				IF CountAO = 0 THEN 
				// code for invalid object address	IOA : return command with invalid data . 
					stTxAsdu := stRxAsdu;
					IF stRxAsdu.info.objAddr = AODB[KK].aObj.obj.info.objAddr THEN
						stTxAsdu.ident.eCOT := eIEC870_COT_UNKNOWN_TYPE; // cause of transfer -> Wrong TYPE for this IoA .  
					ELSE
						stTxAsdu.ident.eCOT := eIEC870_COT_UNKNOWN_OBJECT_ADDRESS; // cause of transfer -> unknown IOA 
					END_IF
					stTxAsdu.ident.bPN :=  TRUE;					
					fbBuffer.TxAddObj(	putObj := stTxAsdu,
										buffer := stBuffer);
					IF NOT fbBuffer.bOk THEN
						// code for buffer overflow
						EXIT; 
					END_IF		 
					EXIT;
				END_IF
				
				
			C_SE_TC_1: // Télévaleurs	
				CountAO := 0 ; 
				FOR KK:=1 TO akuoPara.iAOnb DO 
					IF stRxAsdu.info.objAddr = AODB[KK].aObj.obj.info.objAddr THEN 
						CountAO := CountAO +1 ; ;
						F_iecCopyStreamToBuffer(ADR(nSCO_Val),SIZEOF(nSCO_Val),stRxAsdu.info.stream);
						// Get value of corresponding byte .
						TempData_bis := MesDword_Old[KK] XOR SHL(MesCmd_old[KK] ,AODB[KK].aObj.cfg.bitOffs )  ; 	// We set to zero here the bits that will be replaced
						TempData_bis := SHL(nSCO_Val AND Mask[KK] , AODB[KK].aObj.cfg.bitOffs) OR TempData_bis ;	// We insert the new bits 
			
						IF NOT IN_Local	THEN				// Permet de mettre à jour la commande que si pas en local
							MEMCPY( destAddr := memory+ULINT_TO_DWORD(AODB[KK].aObj.cfg.byteOffs) , srcAddr := ADR(TempData_bis) , n := nBytesRead[KK]);
							MesCmd := nSCO_Val AND Mask[KK] ;
					
						ELSE
							nSCO_Val := MesCmd_old[KK] ;
						END_IF	
					
						// create activation confirmation asdu
						stTxAsdu := stRxAsdu;
						F_iecCopyStreamToBufferByOffset(ADR(nSCO_Val),SIZEOF(nSCO_Val),0,stTxAsdu.info.stream);// Permet de mettre à jour que si pas en local	
						stTxAsdu.ident.eCOT := eIEC870_COT_ACT_CON; 				//cause of transfer -> activation confirmation
						
						IF IN_Local THEN
							stTxAsdu.ident.bPN :=  TRUE;
						ELSE 
							stTxAsdu.ident.bPN := FALSE;
						END_IF						
						
						fbBuffer.TxAddObj(	putObj := stTxAsdu,	buffer := stBuffer);
						IF NOT fbBuffer.bOk THEN
							// code for buffer overflow
							EXIT; 
						END_IF
						
						IF NOT IN_Local THEN
							stTxAsdu := stRxAsdu;
							stTxAsdu.ident.eCOT := eIEC870_COT_ACT_TERM; // cause of transfer -> activation termination
							stTxAsdu.ident.bPN := FALSE;
							fbBuffer.TxAddObj(	putObj := stTxAsdu,	buffer := stBuffer);
							IF NOT fbBuffer.bOk THEN
								// code for buffer overflow
								EXIT; 
							END_IF				
						END_IF
						
					END_IF
				END_FOR
				
				IF CountAO = 0 THEN 
				// code for invalid object address	IOA : return command with invalid data . 
					stTxAsdu := stRxAsdu;
					IF stRxAsdu.info.objAddr = AODB[KK].aObj.obj.info.objAddr THEN
						stTxAsdu.ident.eCOT := eIEC870_COT_UNKNOWN_TYPE; // cause of transfer -> Wrong TYPE for this IoA .  
					ELSE
						stTxAsdu.ident.eCOT := eIEC870_COT_UNKNOWN_OBJECT_ADDRESS; // cause of transfer -> unknown IOA 
					END_IF
					stTxAsdu.ident.bPN :=  TRUE;					
					fbBuffer.TxAddObj(	putObj := stTxAsdu,
										buffer := stBuffer);
					IF NOT fbBuffer.bOk THEN
						// code for buffer overflow
						EXIT; 
					END_IF		 
					EXIT;
				END_IF
			
			C_CS_NA_1: 
				// clock synchronisation
				F_iecCopyStreamToBuffer(ADR(tActTime),SIZEOF(tActTime),stRxAsdu.info.stream);	
	
				// create clock sync confirmation asdu
				stTxAsdu := stRXAsdu;
				stTxAsdu.ident.eCOT := eIEC870_COT_ACT_CON; // cause of transfer -> activation confirmation
				fbBuffer.TxAddObj(	putObj := stTxAsdu,
									buffer := stBuffer);
				IF NOT fbBuffer.bOk THEN
					// code for buffer overflow
					EXIT; 
				END_IF
				// set local computer time
				fbsetLocalTime( START	:= TRUE,
								NETID	:= '', 
								TIMESTR	:= CP56Time2a_TO_SYSTEMTIME(tActTime,20) );
				fbsetLocalTime( START	:= FALSE);
		ELSE
				// code for invalid asdu types 
				stTxAsdu := stRxAsdu;
				stTxAsdu.ident.eCOT := eIEC870_COT_UNKNOWN_TYPE; // cause of transfer -> unknown Type ASDU 
				stTxAsdu.ident.bPN :=  TRUE;					
				fbBuffer.TxAddObj(	putObj := stTxAsdu,
									buffer := stBuffer);
				IF NOT fbBuffer.bOk THEN
					// code for buffer overflow
					EXIT; 
				END_IF		
			
			EXIT;
		END_CASE
	END_IF

UNTIL NOT fbBuffer.bOk // RX fifo is empty
END_REPEAT
END_METHOD

END_FUNCTION_BLOCK

// ---- 00_FunctionsBlocks/Common/AlarmManagement/FB_DetectFlicker.TcPOU
FUNCTION_BLOCK FB_DetectFlicker
// Detect if a booleean variable is flickering 

VAR_INPUT
	IN_VAR			: BOOL;						// Boolean input to analyze
	IN_Window		: TIME := T#5S;				// Time Window during which I check the number of value change
	IN_Count		: UINT;						// Maximum number of change for the tiume duration 

END_VAR
VAR_OUTPUT
	OUT_bFlicker		: BOOL;					// Value is considered as flickering
END_VAR
VAR
	COUNT 			: CTU ; 
	TON				: TON ; 
END_VAR

TON(IN:= TRUE , PT:= IN_Window ) ; 

IF COUNT.CV > IN_Count THEN 
	OUT_bFlicker := TRUE ; 
ELSIF COUNT.CV < IN_Count AND TON.Q THEN  
	OUT_bFlicker := FALSE ; 
END_IF	
	
COUNT(CU:= IN_VAR , PV:= 1000 , RESET:=TON.Q)  ; 

IF TON.Q THEN 
	TON(IN:= FALSE ) ; 
END_IF

END_FUNCTION_BLOCK

// ---- 00_FunctionsBlocks/Beckhoff/Communication/ModbusRTU/Sample_ModbusRTU.TcPOU
PROGRAM Sample_ModbusRTU
VAR
	ModbusRTU				: FB_ModbusRTU;
	MesBlock				: ARRAY[1..8] OF ARRAY[1..120] OF WORD;	
	AX_Addr					: ARRAY[1..8] OF UINT 	:= [1,		1,		1,		1,		1, 		1, 		1, 		1];
	AX_Qty					: ARRAY[1..8] OF UINT	:= [1,		1,		1,		1,		1, 		1, 		1, 		1];
	AX_UnitId				: ARRAY[1..8] OF BYTE	:= [1,		1,		1,		1,		1, 		1, 		1, 		1];
	AX_Function				: ARRAY[1..8] OF UINT	:= [1,		2,		3,		4,		5, 	 	6, 	 	15, 	16];	
	AX_Priority				: ARRAY[1..8] OF UINT	:= [1,		1,		1,		1,		1, 	 	1, 	 	1, 		1 ];
	AX_bStart				: ARRAY[1..8] OF BOOL;
	MbStruct				: ARRAY[1..8] OF Struct_InputRTU;	
	
	KK: INT;
END_VAR

ModbusRTU();

FOR KK := 1 TO 8 DO 
	MbStruct[KK].InBuffer := ADR(MesBlock[KK]);
	MbStruct[KK].InFunction := AX_Function[KK];
	MbStruct[KK].InQuantity := AX_Qty[KK];
	MbStruct[KK].InStartAddr := AX_Addr[KK];
	MbStruct[KK].InUnitID := AX_UnitId[KK];
END_FOR


IF CalLocalTimeStruct.wSecond MOD 5 = 0 THEN
	FOR KK := 1 TO 8 DO
		IF AX_bStart[KK] THEN
			ModbusRTU.M_AddAction_FIFO(InStruct := MbStruct[KK], InPriority := AX_Priority[KK]);
		END_IF
	END_FOR
	
END_IF

END_PROGRAM

// ---- 00_FunctionsBlocks/Beckhoff/Communication/ModbusTCP/FB_ModbusReadCoils.TcPOU
FUNCTION_BLOCK FB_ModbusReadCoils
////////////////// 
// Read Modbus TCP/IP on Rising Edge of Trigger ClockRead. Returns alarm and stop modbus Read after three consecutive Modbus attempts that failed. 
//////////////////

VAR_INPUT
	
	// Modbus ReadRegs FB inputs
	pDestAddr 	: POINTER TO BYTE ; // Pointer to variable in which the read data have to be stored
	sIPAddr 	: STRING(15);		// Modbus server device IP adress
	tTimeout 	: TIME;				// Timeout
	nTcpPort 	: UINT;
	nQuantity 	: WORD;				// Quantity of words to be read
	nMBAddr 	: WORD ;			// Starting Register adress
	
	cbLength 	: UDINT;			// Length of variable to host the read data
	nUnitID 	: BYTE;				// Unit ID in case of serial connexion after modbus server. Usually equals to 1
	
	ClockRead	: BOOL; 			// Rising Edge Modbus Trigger
	Reset		: BOOL; 			// Reset Trigger to clean alarm and counter.
	
END_VAR

VAR_OUTPUT
	ErrorId			: UDINT;	// Error Id returned by FB ( see ADS error Code ) . 
	
	Busy			: BOOL ;	// FB busy to proceed command
	ModbusReadAlarm	: BOOL; 	// Alarm if three modbus attempt failed.
	OUT_NbRead		: UDINT;
END_VAR

VAR
	R_TRIG 				: R_TRIG; 			// Rising edge detection for the trigger.
	FB_MBReadCoils 		: FB_MBReadCoils; 	// Multiple registers reading
	
	Step				: INT; 				// Grafcet step
	AlarmCounter		: INT; 				// Alarm Counter. Incremennted if modbus errOR  Alarm if counter =3 , resetable.  

	
END_VAR

// ALARM MANAGEMENT //

	IF AlarmCounter=3 THEN 
		ModbusReadAlarm 	:=TRUE;
		
	ELSE
		ModbusReadAlarm := FALSE;
		ErrorId			:= 0;
		
	END_IF


// MODBUS SEQUENCE //
CASE Step OF 
	0:
		R_TRIG(CLK :=ClockRead);
		
		IF R_TRIG.Q THEN 
			Step :=1;
			Busy := TRUE;
			OUT_NbRead := 0;
		END_IF
	1:
	   FB_MBReadCoils(
	  			sIPAddr:= sIPAddr , 
				nTCPPort:= nTcpPort ,
				nUnitID:= nUnitID,
				nQuantity:= nQuantity,
				nMBAddr:= nMBAddr, 
				cbLength:= cbLength, 
				pDestAddr:= pDestAddr, 
				bExecute:= TRUE,
				tTimeout:= tTimeout,
				cbRead => OUT_NbRead
				);
				
		IF NOT FB_MBReadCoils.bBusy AND NOT FB_MBReadCoils.bError THEN
			FB_MBReadCoils(bExecute:= FALSE);
			AlarmCounter	:=0; // Reset counter after successful modbus read. 
			Step 			:=0;
			Busy := FALSE;
		ELSIF NOT FB_MBReadCoils.bBusy AND FB_MBReadCoils.bError THEN
			FB_MBReadCoils(bExecute:= FALSE);
			AlarmCounter 	:= MIN(AlarmCounter+1,3) ; 
			ErrorId			 :=FB_MBReadCoils.nErrId;
			Step 			:=0;
			Busy := FALSE;
		END_IF
		
END_CASE

// RESET //
	IF Reset THEN 
			AlarmCounter 		:= 0 ; 
			ErrorId 			:= 0 ; 
			ModbusReadAlarm 	:=FALSE;
			Reset 				:= FALSE;
			FB_MBReadCoils		(bExecute := FALSE);
	END_IF

// BUSY //

END_FUNCTION_BLOCK

// ---- 00_FunctionsBlocks/Beckhoff/Communication/ModbusTCP/FB_ModbusReadInput.TcPOU
FUNCTION_BLOCK FB_ModbusReadInput
////////////////// 
// Read Modbus TCP/IP on Rising Edge of Trigger ClockRead. Returns alarm and stop modbus Read after three consecutive Modbus attempts that failed. 
//////////////////

VAR_INPUT
	
	// Modbus ReadRegs FB inputs
	pDestAddr 	: POINTER TO BYTE ; // Pointer to variable in which the read data have to be stored
	sIPAddr 	: STRING(15);		// Modbus server device IP adress
	tTimeout 	: TIME;				// Timeout
	nTcpPort 	: UINT;
	nQuantity 	: WORD;				// Quantity of words to be read
	nMBAddr 	: WORD ;			// Starting Register adress
	
	cbLength 	: UDINT;			// Length of variable to host the read data
	nUnitID 	: BYTE;				// Unit ID in case of serial connexion after modbus server. Usually equals to 1
	
	ClockRead	: BOOL; 			// Rising Edge Modbus Trigger
	Reset		: BOOL; 			// Reset Trigger to clean alarm and counter.
	
END_VAR

VAR_OUTPUT
	ErrorId			: UDINT;	// Error Id returned by FB ( see ADS error Code ) . 
	
	Busy			: BOOL ;	// FB busy to proceed command
	ModbusReadAlarm	: BOOL; 	// Alarm if three modbus attempt failed.
	OUT_NbRead		: UDINT;
END_VAR

VAR
	R_TRIG 				: R_TRIG; 			// Rising edge detection for the trigger.
	FB_MBReadInputs 		: FB_MBReadInputs; 	// Multiple registers reading
	
	Step				: INT; 				// Grafcet step
	AlarmCounter		: INT; 				// Alarm Counter. Incremennted if modbus errOR  Alarm if counter =3 , resetable.  

	
END_VAR

// ALARM MANAGEMENT //

	IF AlarmCounter=3 THEN 
		ModbusReadAlarm 	:=TRUE;
		
	ELSE
		ModbusReadAlarm := FALSE;
		ErrorId			:= 0;
		
	END_IF


// MODBUS SEQUENCE //
CASE Step OF 
	0:
		R_TRIG(CLK :=ClockRead);
		
		IF R_TRIG.Q THEN 
			Step :=1;
			Busy := TRUE;
			OUT_NbRead := 0;
		END_IF
	1:
	   FB_MBReadInputs(
	  			sIPAddr:= sIPAddr , 
				nTCPPort:= nTcpPort ,
				nUnitID:= nUnitID,
				nQuantity:= nQuantity,
				nMBAddr:= nMBAddr, 
				cbLength:= cbLength, 
				pDestAddr:= pDestAddr, 
				bExecute:= TRUE,
				tTimeout:= tTimeout,
				cbRead => OUT_NbRead
				);
				
		IF NOT FB_MBReadInputs.bBusy AND NOT FB_MBReadInputs.bError THEN
			FB_MBReadInputs(bExecute:= FALSE);
			AlarmCounter	:=0; // Reset counter after successful modbus read. 
			Step 			:=0;
			Busy := FALSE;
		ELSIF NOT FB_MBReadInputs.bBusy AND FB_MBReadInputs.bError THEN
			FB_MBReadInputs(bExecute:= FALSE);
			AlarmCounter 	:= MIN(AlarmCounter+1,3) ; 
			ErrorId			 :=FB_MBReadInputs.nErrId;
			Step 			:=0;
			Busy := FALSE;
		END_IF
		
END_CASE

// RESET //
	IF Reset THEN 
			AlarmCounter 		:= 0 ; 
			ErrorId 			:= 0 ; 
			ModbusReadAlarm 	:=FALSE;
			Reset 				:= FALSE;
			FB_MBReadInputs		(bExecute := FALSE);
	END_IF

// BUSY //

END_FUNCTION_BLOCK

// ---- 00_FunctionsBlocks/Beckhoff/Communication/ModbusTCP/FB_ModbusWriteMultipleCoils.TcPOU
FUNCTION_BLOCK FB_ModbusWriteMultipleCoils
////////////////// 
// Write Modbus TCP/IP on Rising Edge of Trigger WriteCommAND  Returns alarm and stop modbus Read after three consecutive Modbus attempts that failed.
// Write two registers 
//////////////////
VAR_INPUT
	// Modbus ReadRegs FB inputs

	pSrcAddr			: POINTER TO BYTE ;
	sIPAddr 			: STRING(15);
	tTimeout 			: TIME;
	nTCPport			: UINT:= 502;		// TCP Port
	nMBAddr 			: WORD ;
	cbLength 			: UDINT ;
	nQuantity			: BYTE ;
	nUnitID 			: BYTE;
	WriteCmd 			: BOOL; 					// Rising Edge Trigger for sending modbus request
	
	Reset				: BOOL; 					// Reset Trigger to clean alarm and counter	
	
END_VAR


VAR_OUTPUT
	ErrorId				: UDINT; 			// Erreur ID returned by FB modbus. Updated every time on error occurs. 
	
	Completed			: BOOL ;			// Modbus Writing is completed 
	Busy				: BOOL ; 			// FB busy to proceed command
	ModbusWriteAlarm	: BOOL; 			// Alarm if three modbus attempt failed.
	
END_VAR
VAR
	R_TRIG 				: R_TRIG; 				// Rising edge detection for the trigger.
	FB_MBWriteCoils		: FB_MBWriteCoils; 		// Multiple registers reading
	
	Step				: INT; 					// Grafcet step
	AlarmCounter		: INT; 					// Alarm Counter. Incremennted if modbus errOR  Alarm if counter =3 , resetable.  
END_VAR

Completed 				:= FALSE ;

// ALARM MANAGEMENT //
IF AlarmCounter=3 THEN
	ModbusWriteAlarm 	:=TRUE;
	
ELSE
	ModbusWriteAlarm 	:= FALSE;
	ErrorId				:= 0;
	
END_IF
	
// MODBUS SEQUENCE //
	CASE Step OF 
		0:
			R_TRIG(CLK :=WriteCmd);
			IF R_TRIG.Q THEN 
				Step :=1;
			END_IF
			
		1:
		   FB_MBWriteCoils(
					sIPAddr:= sIPAddr , 
					nTCPPort:= nTCPport ,
					nUnitID:= nUnitID,
					nQuantity:= nQuantity,
					nMBAddr:= nMBAddr, 
					cbLength:= cbLength, 
					pSrcAddr:= pSrcAddr, 
					bExecute:= TRUE,
					tTimeout:= tTimeout
					);
					
			IF NOT FB_MBWriteCoils.bBusy AND NOT FB_MBWriteCoils.bError THEN
				FB_MBWriteCoils(bExecute:= FALSE);
				AlarmCounter		:=0; // Reset counter after successful modbus read. 
				Step 				:=0;
				Completed 			:= TRUE ;
				
			ELSIF NOT FB_MBWriteCoils.bBusy AND FB_MBWriteCoils.bError THEN
				FB_MBWriteCoils(bExecute:= FALSE);
				AlarmCounter 		:=MIN(AlarmCounter+1,3) ; 
				ErrorId			 	:=FB_MBWriteCoils.nErrId;
				Step 				:=0;
				
			END_IF
			
	END_CASE

// RESET //	
	IF Reset THEN 
			AlarmCounter 	:= 0 ; 
			ErrorId 		:= 0 ; 
	END_IF	
	
// BUSY //
	Busy 					:= FB_MBWriteCoils.bBusy ;

END_FUNCTION_BLOCK

// ---- 00_FunctionsBlocks/Beckhoff/Communication/ModbusTCP/FB_ModbusWriteSingleCoil.TcPOU
FUNCTION_BLOCK FB_ModbusWriteSingleCoil
////////////////// 
// Write Modbus TCP/IP on Rising Edge of Trigger WriteCommAND  Returns alarm and stop modbus Read after three consecutive Modbus attempts that failed.
// Write two registers 
//////////////////
VAR_INPUT
	// Modbus ReadRegs FB inputs
	bValue 				: BOOL;
	sIPAddr 			: STRING(15);
	tTimeout 			: TIME;
	nTCPport			: UINT:= 502;		// TCP Port
	nMBAddr 			: WORD ;
	nUnitID 			: BYTE;
	WriteCmd 			: BOOL; 					// Rising Edge Trigger for sending modbus request
	
	Reset				: BOOL; 					// Reset Trigger to clean alarm and counter	
	
END_VAR


VAR_OUTPUT
	ErrorId				: UDINT; 			// Erreur ID returned by FB modbus. Updated every time on error occurs. 
	
	Completed			: BOOL ;			// Modbus Writing is completed 
	Busy				: BOOL ; 			// FB busy to proceed command
	ModbusWriteAlarm	: BOOL; 			// Alarm if three modbus attempt failed.
	
END_VAR
VAR
	R_TRIG 				: R_TRIG; 				// Rising edge detection for the trigger.
	FB_MBWriteSingleCoil: FB_MBWriteSingleCoil; 		// Multiple registers reading
	
	Step				: INT; 					// Grafcet step
	AlarmCounter		: INT; 					// Alarm Counter. Incremennted if modbus errOR  Alarm if counter =3 , resetable.  
	wValue				: WORD;
END_VAR

Completed 				:= FALSE ;

// ALARM MANAGEMENT //
IF AlarmCounter=3 THEN
	ModbusWriteAlarm 	:=TRUE;
	
ELSE
	ModbusWriteAlarm 	:= FALSE;
	ErrorId				:= 0;
	
END_IF

IF bValue THEN
	wValue := 16#FF00;
ELSE
	wValue := 16#0000;
END_IF
	
// MODBUS SEQUENCE //
	CASE Step OF 
		0:
			R_TRIG(CLK :=WriteCmd);
			IF R_TRIG.Q THEN 
				Step :=1;
			END_IF
			
		1:
		   FB_MBWriteSingleCoil
			(
				sIPAddr:= sIPAddr ,
				nValue := wValue,
				nTCPPort:= nTCPport ,
				nUnitID:= nUnitID,
				nMBAddr:= nMBAddr, 
				bExecute:= TRUE,
				tTimeout:= tTimeout
			);
					
			IF NOT FB_MBWriteSingleCoil.bBusy AND NOT FB_MBWriteSingleCoil.bError THEN
				FB_MBWriteSingleCoil(bExecute:= FALSE);
				AlarmCounter		:=0; // Reset counter after successful modbus read. 
				Step 				:=0;
				Completed 			:= TRUE ;
				
			ELSIF NOT FB_MBWriteSingleCoil.bBusy AND FB_MBWriteSingleCoil.bError THEN
				FB_MBWriteSingleCoil(bExecute:= FALSE);
				AlarmCounter 		:=MIN(AlarmCounter+1,3) ; 
				ErrorId			 	:=FB_MBWriteSingleCoil.nErrId;
				Step 				:=0;
				
			END_IF
			
	END_CASE

// RESET //	
	IF Reset THEN 
			AlarmCounter 	:= 0 ; 
			ErrorId 		:= 0 ; 
	END_IF	
	
// BUSY //
	Busy 					:= FB_MBWriteSingleCoil.bBusy ;

END_FUNCTION_BLOCK

// ---- 00_FunctionsBlocks/Beckhoff/Communication/ModbusTCP/FB_ModbusWriteSingleRegister.TcPOU
FUNCTION_BLOCK FB_ModbusWriteSingleRegister
////////////////// 
// Write Modbus TCP/IP on Rising Edge of Trigger WriteCommAND  Returns alarm and stop modbus Read after three consecutive Modbus attempts that failed.
// Write two registers 
//////////////////
VAR_INPUT
	// Modbus ReadRegs FB inputs

	InputWord			: WORD ;
	sIPAddr 			: STRING(15);
	tTimeout 			: TIME;
	nTCPport			: UINT:= 502;		// TCP Port
	nMBAddr 			: WORD ;
	cbLength 			: UDINT ;
	nQuantity			: BYTE ;
	nUnitID 			: BYTE;
	WriteCmd 			: BOOL; 					// Rising Edge Trigger for sending modbus request
	
	Reset				: BOOL; 					// Reset Trigger to clean alarm and counter	
	
END_VAR


VAR_OUTPUT
	ErrorId						: UDINT; 			// Erreur ID returned by FB modbus. Updated every time on error occurs. 
	                    		
	Completed					: BOOL ;			// Modbus Writing is completed 
	Busy						: BOOL ; 			// FB busy to proceed command
	ModbusWriteAlarm			: BOOL; 			// Alarm if three modbus attempt failed.
	
END_VAR
VAR
	R_TRIG 						: R_TRIG; 				// Rising edge detection for the trigger.
	MBWriteSingleReg 		: FB_MBWriteSingleReg; 		// Multiple registers reading
	
	Step						: INT; 					// Grafcet step
	AlarmCounter				: INT; 					// Alarm Counter. Incremennted if modbus errOR  Alarm if counter =3 , resetable.  
END_VAR

Completed 				:= FALSE ;

// ALARM MANAGEMENT //
IF AlarmCounter=3 THEN
	ModbusWriteAlarm 	:=TRUE;
	
ELSE
	ModbusWriteAlarm 	:= FALSE;
	ErrorId				:= 0;
	
END_IF
	
// MODBUS SEQUENCE //
	CASE Step OF 
		0:
			R_TRIG(CLK :=WriteCmd);
			IF R_TRIG.Q THEN 
				Step :=1;
			END_IF
			
		1:
		   MBWriteSingleReg(
			   		nValue := InputWord,
					sIPAddr:= sIPAddr , 
					nTCPPort:= nTCPport ,
					nUnitID:= nUnitID,
					nMBAddr:= nMBAddr, 
					bExecute:= TRUE,
					tTimeout:= tTimeout
					);
					
			IF NOT MBWriteSingleReg.bBusy AND NOT MBWriteSingleReg.bError THEN
				MBWriteSingleReg(bExecute:= FALSE);
				AlarmCounter		:=0; // Reset counter after successful modbus read. 
				Step 				:=0;
				Completed 			:= TRUE ;
				
			ELSIF NOT MBWriteSingleReg.bBusy AND MBWriteSingleReg.bError THEN
				MBWriteSingleReg(bExecute:= FALSE);
				AlarmCounter 		:=MIN(AlarmCounter+1,3) ; 
				ErrorId			 	:=MBWriteSingleReg.nErrId;
				Step 				:=0;
				
			END_IF
			
	END_CASE

// RESET //	
	IF Reset THEN 
			AlarmCounter 	:= 0 ; 
			ErrorId 		:= 0 ; 
			Reset			:= FALSE;
			MBWriteSingleReg(bExecute := FALSE);
	END_IF	
	
// BUSY //
	Busy 					:= MBWriteSingleReg.bBusy ;

END_FUNCTION_BLOCK

// ---- 00_FunctionsBlocks/Beckhoff/Database/CheckConfig.TcPOU
PROGRAM CheckConfig
VAR_INPUT
		IN_Start				: BOOL := TRUE;
		ParamInitWait			: TIME := T#5S;
END_VAR
VAR_OUTPUT
		OUT_aDBConfig         		: ARRAY[0..MAX_CONFIGURATIONS] OF ST_ConfigDB;
		OUT_Busy					: BOOL;
		OUT_Error					: BOOL;
		OUT_Result					: INT;
END_VAR
VAR
	// CheckConfig    
		TON_CheckConfig				: TON;      		
		TrigCheckConfig				: R_TRIG;
		TrigInit					: F_TRIG;
		RS_CheckConfig				: RS;
		                    		
		ConfigTcDBSrvEvt  			: FB_ConfigTcDBSrvEvt(sNetId := '', tTimeout:=T#5S);
		                    		
		aAutoGrpConfig    			: ARRAY[0..MAX_CONFIGURATIONS] OF ST_ConfigAutoLogGrp;
		AX_NameBase					: ARRAY[0..MAX_CONFIGURATIONS] OF T_MaxString;
		AX_hDBID					: ARRAY[0..MAX_CONFIGURATIONS] OF BOOL;
		AX_hDBIDNull				: ARRAY[0..MAX_CONFIGURATIONS] OF BOOL;
		                    		
		nDbCount          			: UDINT;
		nAutoGrpCount     			: UDINT;

		KK : UDINT;
END_VAR

TON_CheckConfig(IN := IN_Start, PT := ParamInitWait);

TrigCheckConfig(CLK := TON_CheckConfig.Q);
RS_CheckConfig(SET := TrigCheckConfig.Q);
IF TrigCheckConfig.Q THEN
	IN_Start := FALSE;
	OUT_Result := 0;
END_IF
IF RS_CheckConfig.Q1 THEN
	
	OUT_Busy := TRUE;
	IF ConfigTcDBSrvEvt.Read(pDBConfig := ADR(OUT_aDBConfig), cbDBConfig := SIZEOF(OUT_aDBConfig), pAutologGrpConfig := ADR(aAutoGrpConfig),
			cbAutoLogGrpConfig := SIZEOF(aAutoGrpConfig),pDBCount := ADR(nDbCount),pAutoLogGrpCount := ADR(nAutoGrpCount)) THEN
		
		IF ConfigTcDBSrvEvt.bError THEN
			OUT_Result := -1;
		ELSE
			FOR KK := 0 TO MAX_CONFIGURATIONS DO
				AX_hDBID[OUT_aDBConfig[KK].hDBID] := OUT_aDBConfig[KK].hDBID <> 0;
				AX_NameBase[KK] :=  OUT_aDBConfig[KK].sName;
			END_FOR
			OUT_Result := 1;
		END_IF  
		RS_CheckConfig(RESET1 := TRUE);
		RS_CheckConfig(RESET1 := FALSE);
		OUT_Busy := FALSE;
		
	END_IF
END_IF

END_PROGRAM

// ---- 00_FunctionsBlocks/Beckhoff/Database/Firebird/Firebird_CreateTables.TcPOU
PROGRAM Firebird_CreateTables
VAR_INPUT
	IN_Start				: BOOL;
	IN_TableNames			: ARRAY[1.. CstNbTables] OF STRING;
	IN_hDBID         		: UDINT;	
END_VAR
VAR_OUTPUT
	OUT_Error				: BOOL;
	OUT_Busy				: BOOL;
	OUT_Result				: INT;
END_VAR
VAR
	Etape					: UINT;
	
	TrigStart				: R_TRIG;
	RsStart					: RS;
	bCreateTable			: BOOL;
	TrigCreateTable			: R_TRIG;
	RsCreateTable			: RS;
	PLCDBCreateEvt 			: FB_PLCDBCreateEvt(sNetID := '', tTimeout := T#5S);
	FirebirdConf			: T_DBConfig_Odbc;
	sExtension				: STRING:= '.db';
	tcMessage    	 		: I_TcMessage;
	
	AX_ColArray				: ARRAY[0..3] OF ST_ColumnInfo;
	
	NumTable				: UINT := 1;
	KK						: UDINT;
END_VAR


AX_ColArray[0].sName := 'TimeStamp';     	AX_ColArray[0].eType := E_ColumnType.DateTime;   	AX_ColArray[0].nLength := 4;    
AX_ColArray[1].sName := 'TimeStamp_Ms';    	AX_ColArray[1].eType := E_ColumnType.Integer;    	AX_ColArray[1].nLength := 4;
AX_ColArray[2].sName := 'ParentId';   		AX_ColArray[2].eType := E_ColumnType.Integer;   	AX_ColArray[2].nLength := 4;
AX_ColArray[3].sName := 'Value';   			AX_ColArray[3].eType := E_ColumnType.Float;   		AX_ColArray[3].nLength := 8;


TrigCreateTable(CLK := IN_Start);
RsCreateTable(SET:= TrigCreateTable.Q);

IF RsCreateTable.Q1 THEN
	OUT_Busy := TRUE;
	IF NumTable <= CstNbTables THEN
		IF PLCDBCreateEvt.Table(hDBID := IN_hDBID, sTableName := IN_TableNames[NumTable],  pTableCfg := ADR(AX_ColArray), cbTableCfg := SIZEOF(AX_ColArray)  ) THEN
			IF PLCDBCreateEvt.bError THEN
				Etape := 255;
				OUT_Error := TRUE;
				OUT_Result := -2;
			ELSE
				IF Numtable = CstNbTables THEN
					IN_Start := FALSE;
					Etape := 0;
					RsCreateTable(RESET1 := TRUE);
					RsCreateTable(RESET1 := FALSE);	
					bCreateTable := FALSE;
					OUT_Result := 1;	
					TrigStart(CLK := FALSE);
					OUT_Busy := FALSE;	
					OUT_Error := FALSE;
					OUT_Result := 1;
				ELSE
					NumTable := NumTable + 1;		
				END_IF
			END_IF
		END_IF
	END_IF
END_IF

IF Etape = 255 THEN
	Etape := 0;
	bCreateTable := FALSE;
	IN_Start := FALSE;
	OUT_Busy := FALSE;	
	RsCreateTable(RESET1 := TRUE);
	RsCreateTable(RESET1 := FALSE);
END_IF

END_PROGRAM

// ---- 00_FunctionsBlocks/Beckhoff/Database/Firebird/Firebird_InsertBuffer.TcPOU
FUNCTION_BLOCK Firebird_InsertBuffer
// Fonctionnement : Tableau de 2000 structures en input. Dès qu'on atteint 1000 structures remplies, décalage de l'espace mémoire
// pour en 1 temps de cycle pour ne pas perdre de données sur le transfert.
VAR CONSTANT
	//CstNbLigneBuffer					: UINT:= 500;
	CstNbLigneBufferMax	 				: DINT:= 1000;
                            			
END_VAR                     			
                            			
VAR_INPUT                   			
	NomTable							: STRING(255) := 'Table100ms';
	IN_Reset							: BOOL;
	IN_Hdbid							: DINT;
	ParamTimeOut						: TIME := T#10s;
END_VAR                     			
                            			
VAR_OUTPUT                  			
	OUT_Error							: BOOL;
	OUT_Busy							: BOOL;
	OUT_Result							: INT;
	Out_Connected						: BOOL;
END_VAR                     			
                            			
VAR                         		
	Etape_main							: UINT:=2;	
	ETAPE								: UINT;
		CstNbLigneBuffer					: UINT:= 500;
	FTrig_TP_Retry						: F_TRIG;                        			
	TrigReset							: R_TRIG;
	TON_Watchdog						: TON ;
	TP_Retry							: TP;
	Tmp_Nb_Buffer						: DINT;
    //myStruct      						: ARRAY[1..CstNbLigneBuffer] OF St_DataHisto;
	//myStructMax    						: ARRAY[1..CstNbLigneBufferMax] OF St_DataHisto;
	StructNull							: St_DataHisto;
                            			
    SQLDatabase1						: FB_SQLDatabaseEvt('',T#10S);
    SQLDatabase2						: FB_SQLDatabaseEvt('',T#10S);
	SQLCommand1							: FB_SQLCommandEvt('',T#10S);
	SQLCommand2							: FB_SQLCommandEvt('',T#10S);
	
	bConnected							: BOOL;              	        	
                            			
	TrameValues							: T_MaxString := ' ([Timestamp],[ParentId],[Value])';
	pPosRequete							: DINT;                		
	RequeteFinale						: ARRAY[1..10000] OF STRING(1000);	
	RequeteFinaleNull					: ARRAY [1..10000] OF STRING(1000);
	
	sTimeStamp							: STRING(255);  
	RequeteEntete						: STRING(1000);
	sInsertValue						: STRING(1000);
	Format								: FB_FormatString;
	                			
	NbElemBuffer						: DINT;
	KK									: DINT;
	                    				
	CmdStart							: BOOL;
	TrigRestartMaxReached				: R_TRIG;
	TrigCmdExec							: R_TRIG;
	TrigStart							: R_TRIG;
	RsStart								: RS;
	                        			
	// AlarmManagement      			
		bBufferMaxFull 					: BOOL;        		
		bInStructNull					: BOOL;
		
	// CONNECT	
		TrigStartConnect				: R_TRIG;	
		RsStartConnect					: RS;
	// DISCONNECT
		TrigStartDisconnect				: R_TRIG;
		RsStartDisconnect				: RS;

		bReconnect						: BOOL;
		FTrig_bReconnect				: F_TRIG;
			
	MesAlarm: BOOL;
	TrigWatchdog : R_TRIG;
	bTest: BOOL;
	FIFO						: FB_DBDatasetFifo_1min;
END_VAR    

VAR_IN_OUT
	
END_VAR


//CmdStart := FIFO.nCount>= CstNbLigneBuffer AND NOT FTrig_TP_Retry.Q;
CmdStart := FIFO.nCount >= 0 AND NOT FTrig_TP_Retry.Q;


TP_Retry(IN := FIFO.nCount >= CstNbLigneBufferMax AND NOT TP_Retry.Q, PT := T#3S);
FTrig_TP_Retry(CLK := TP_Retry.Q);

TrigReset(CLK := IN_Reset OR TON_Watchdog.Q);
IF TrigReset.Q THEN
	FIFO.A_Reset();
END_IF

TrigStart(CLK := CmdStart);
IF TrigStart.Q THEN
	ETAPE := 1;
END_IF


RsStart(SET := TrigStart.Q);
IF RsStart.Q1 THEN
	RequeteEntete :=  concat(concat(' INSERT INTO "',NomTable),'" ');
END_IF
		
CASE ETAPE OF
		
	1: // CONNECTED
		IF SQLDatabase1.CreateCmd(pSQLCommand := ADR(SQLCommand1)) THEN 
			IF NOT SQLDatabase1.bError THEN
				MEMCPY(srcAddr:= ADR(RequeteEntete), destAddr := ADR(requeteFinale), n:= SIZEOF(RequeteEntete));
				pPosRequete := LEN(STR := RequeteEntete);
				Tmp_Nb_Buffer :=UDINT_TO_DINT(FIFO.nCount -1);
				FOR KK:= 1 TO MIN(Tmp_Nb_Buffer,CstNbLigneBuffer-1) DO
					fifo.A_Get();
					sTimeStamp	:=  SYSTEMTIME_TO_STRING(fifo.Out.Timestamp);
					Format(sFormat := 'select $'%s$',%.4d,%5.2f FROM RDB$$DATABASE UNION ALL ', arg1 := F_STRING(sTimeStamp),arg2:= F_DINT(fifo.out.ParentId), arg3:= F_LREAL(fifo.out.Value), arg5:= F_STRING(NomTable), sOut=>sInsertValue);
					MEMCPY(srcAddr:= ADR(sInsertValue), destAddr := ADR(requeteFinale)+DINT_TO_DWORD(pPosRequete), n:= SIZEOF(sInsertValue));
					pPosRequete:= pPosRequete + LEN(STR := sInsertValue);
					fifo.A_Remove();
				END_FOR
				fifo.A_Get();
				sTimeStamp	:= SYSTEMTIME_TO_STRING(fifo.Out.Timestamp);
				Format(sFormat := 'select $'%s$',%.4d,%5.2f FROM RDB$$DATABASE;', arg1 := F_STRING(sTimeStamp),arg2:= F_DINT(fifo.out.ParentId), arg3:= F_LREAL(fifo.out.Value), sOut=>sInsertValue);
				MEMCPY(srcAddr:= ADR(sInsertValue), destAddr := ADR(requeteFinale)+DINT_TO_DWORD(pPosRequete), n:= SIZEOF(sInsertValue));
				fifo.A_Remove();
				IF Tmp_Nb_Buffer > 0 THEN
					ETAPE := Etape_main;
				END_IF
			ELSIF SQLDatabase1.bError THEN
				ETAPE := 255;
			END_IF
		END_IF
	2:

		IF SQLCommand1.Execute(pSQLCmd := ADR(RequeteFinale), cbSQLCmd := SIZEOF(Requetefinale))THEN
			
			IF  NOT SQLCommand1.bError THEN
				ETAPE := 4;
			ELSIF SQLCommand1.bError THEN
				ETAPE := 255;
			END_IF
		END_IF

	4:
		IF NOT SQLDatabase1.bError THEN
			
			RequeteFinale := RequeteFinaleNull;
			
			//RequeteFinale := '';
			Tmp_Nb_Buffer := MIN(UDINT_TO_DINT(FIFO.nCount),CstNbLigneBuffer);
			//FOR KK:= 1 TO Tmp_Nb_Buffer DO
			//	fifo.A_Remove();
			//END_FOR
			TrigStart(CLK := FALSE);
			RsStart(RESET1 := TRUE);
			RsStart(RESET1 := FALSE);
			TrigCmdExec(CLK := FALSE);
			CmdStart := FALSE;
			Etape := 0;
			OUT_Error := FALSE;
		ELSE 
			ETAPE := 255;
		END_IF
	255: 
		RequeteFinale := RequeteFinaleNull;

		SQLCommand1 := SQLCommand2;
		SQLDatabase1 := SQLDatabase2;
		OUT_Error := TRUE;
		RsStart(RESET1 := TRUE);
		RsStart(RESET1 := FALSE);
		TrigCmdExec(CLK := FALSE);
		CmdStart := FALSE;
		ETAPE := 0;
END_CASE

METHOD M_AddLine : BOOL
VAR_INPUT
	InStruct			: St_DataHisto;
END_VAR

VAR
	InsStruct: St_DataHisto;
END_VAR
fifo.in := InStruct;
fifo.A_Add();
END_METHOD

METHOD M_AlarmManager : BOOL
VAR_INPUT
	AlarmCode : WORD;
	
END_VAR


AlarmCode.0 := bBufferMaxFull;
AlarmCode.1 := bInStructNull;
END_METHOD

METHOD M_Connect : BOOL

VAR_OUTPUT
END_VAR
VAR_INPUT
	IN_hDBID				: DINT;
	IN_Start				: BOOL;
END_VAR
TrigStartConnect(CLK := IN_Start);
RsStartConnect(SET := TrigStartConnect.Q);
IF RsStartConnect.Q1 THEN
	IF SQLDatabase1.Connect(hDBID := IN_hDBID) THEN;
		RsStartConnect(RESET1 := TRUE);
		RsStartConnect(RESET1 := FALSE);
		bReconnect := FALSE;
	END_IF
END_IF

Out_Connected := SQLDatabase1.bConnected;
END_METHOD

METHOD M_Disconnect : BOOL
VAR_INPUT
END_VAR
VAR_INPUT
	IN_Start				: BOOL;
END_VAR
TrigStartDisconnect(CLK := IN_Start);
RsStartDisconnect(SET := TrigStartDisconnect.Q);
IF RsStartDisconnect.Q1 THEN
	FIFO.A_Reset();
	IF SQLDatabase1.Disconnect() THEN;
		RsStartDisconnect(RESET1 := TRUE);
		RsStartDisconnect(RESET1 := FALSE);
	END_IF
END_IF

Out_Connected := SQLDatabase1.bConnected;
END_METHOD

METHOD M_Init

VAR
	LL	: SINT;
	KK 	: SINT;
END_VAR
//Initialisation BUFFER
	//Buffer pour la lecture des sms
	FIFO.A_Reset();
	FIFO.A_Add();
	FIFO.A_Get();
	FIFO.A_Remove();
END_METHOD

END_FUNCTION_BLOCK

// ---- 00_FunctionsBlocks/Beckhoff/Fifo/FB_DBDatasetFifo_1min.TcPOU
FUNCTION_BLOCK FB_DBDatasetFifo_1min
VAR_INPUT
    bOverwrite : BOOL;
    In         : St_DataHisto_Epoch;
END_VAR
VAR_OUTPUT
    bOk        : BOOL;
    nCount     : UDINT;
    nLoad      : UDINT;
    Out        : St_DataHisto_Epoch;
END_VAR
VAR
    arrBuffer  : ARRAY[0..Max_buffer_size_G] OF BYTE; (* Buffer memory used by FB_MemRingBuffer function block *)
    fbBuffer   : FB_MemRingBuffer;
END_VAR

ACTION A_Add:
fbBuffer.A_AddTail(pWrite := ADR(in),
						   cbWrite:=SIZEOF(in),
						   pBuffer:=ADR(arrBuffer),
						   cbBuffer:=SIZEOF(arrBuffer),
						   bOK=>bOK,
						   nCount =>nCount);
IF NOT bOK THEN 
	IF bOverwrite THEN
		fbBuffer.A_RemoveHead();(*remove one oldest entry*)
		fbBuffer.A_AddTail(bOK => bOk,nCount => nCount);
	END_IF
END_IF

nload := (fbbuffer.cbSize * 100)/(Max_buffer_size_G);
END_ACTION

ACTION A_Get:
fbBuffer.A_GetHead(pWrite := ADR(out),
						   cbWrite:=SIZEOF(out),
						   pBuffer:=ADR(arrBuffer),
						   cbBuffer:=SIZEOF(arrBuffer),
						   bOK=>bOK,
						   nCount =>nCount);
nload := (fbbuffer.cbSize * 100)/(Max_buffer_size_G);
END_ACTION

ACTION A_Remove:
fbBuffer.A_RemoveHead(pRead:=ADR(out),
						cbRead:=SIZEOF(out),
						pBuffer:=ADR(arrBuffer),
						cbBuffer:=SIZEOF(arrBuffer),
						bOK=>bOK,
						nCount =>nCount);
nload := (fbbuffer.cbSize * 100)/(Max_buffer_size_G);
END_ACTION

ACTION A_Reset:
MEMSET(ADR(arrBuffer),0,SIZEOF(arrBuffer)); (*reset internal buffer*)
fbBuffer.A_Reset(bOK=>bOK,nCount=>ncount);
nload := (fbbuffer.cbSize * 100)/(Max_buffer_size_G);
END_ACTION

END_FUNCTION_BLOCK

// ---- 00_FunctionsBlocks/Beckhoff/Database/Firebird/Firebird_InsertBuffer_vEpoch.TcPOU
FUNCTION_BLOCK Firebird_InsertBuffer_vEpoch
// Fonctionnement : Tableau de 2000 structures en input. Dès qu'on atteint 1000 structures remplies, décalage de l'espace mémoire
// pour en 1 temps de cycle pour ne pas perdre de données sur le transfert.
VAR CONSTANT
	//CstNbLigneBuffer					: UINT:= 500;
	CstNbLigneBufferMax	 				: DINT:= 1000;
                            			
END_VAR                     			
                            			
VAR_INPUT                   			
	NomTable							: STRING(255) := 'Table100ms';
	IN_Reset							: BOOL;
	IN_Hdbid							: DINT;
	ParamTimeOut						: TIME := T#10s;
END_VAR                     			
                            			
VAR_OUTPUT                  			
	OUT_Error							: BOOL;
	OUT_Busy							: BOOL;
	OUT_Result							: INT;
	OUT_Connected						: BOOL;
END_VAR                     			
                            			
VAR                         			
	ETAPE								: UINT;
	CstNbLigneBuffer					: UINT:= 250;
	
	FTrig_TP_Retry						: F_TRIG;                        			
	TrigReset							: R_TRIG;
	TON_Watchdog						: TON ;
	TP_Retry							: TP;
	Tmp_Nb_Buffer						: DINT;
	StructNull							: St_DataHisto;
                            			
    SQLDatabase1						: FB_SQLDatabaseEvt('',T#10S);
    SQLDatabase2						: FB_SQLDatabaseEvt('',T#10S);
	SQLCommand1							: FB_SQLCommandEvt('',T#10S);
	SQLCommand2							: FB_SQLCommandEvt('',T#10S);
	
	bConnected							: BOOL;              	        	
                            			
	TrameValues							: T_MaxString := ' ([Timestamp],[ParentId],[Value])';
	pPosRequete							: DINT;                		
	RequeteFinale						: ARRAY[1..1000] OF STRING(1000);	
	RequeteFinaleNull					: ARRAY [1..1000] OF STRING(1000);
	
	sTimeStamp							: STRING(255);  
	RequeteEntete						: STRING(1000);
	sInsertValue						: STRING(1000);
	Format								: FB_FormatString;
	                			
	NbElemBuffer						: DINT;
	KK									: DINT;
	                    				
	CmdStart							: BOOL;
	TrigRestartMaxReached				: R_TRIG;
	TrigCmdExec							: R_TRIG;
	TrigStart							: R_TRIG;
	RsStart								: RS;
	                        			
	// AlarmManagement      			
		bBufferMaxFull 					: BOOL;        		
		bInStructNull					: BOOL;
		
	// CONNECT	
		TrigStartConnect				: R_TRIG;	
		RsStartConnect					: RS;
	// DISCONNECT
		TrigStartDisconnect				: R_TRIG;
		RsStartDisconnect				: RS;

		bReconnect						: BOOL;
		FTrig_bReconnect				: F_TRIG;
			
	MesAlarm: BOOL;
	TrigWatchdog : R_TRIG;
	bTest: BOOL;
	FIFO						: FB_DBDatasetFifo_1min;
END_VAR    

VAR_IN_OUT
	
END_VAR


//CmdStart := FIFO.nCount>= CstNbLigneBuffer AND NOT FTrig_TP_Retry.Q;
CmdStart := FIFO.nCount > 0 ;//AND NOT FTrig_TP_Retry.Q;


TP_Retry(IN := FIFO.nCount >= CstNbLigneBufferMax AND NOT TP_Retry.Q, PT := T#3S);
FTrig_TP_Retry(CLK := TP_Retry.Q);

TrigReset(CLK := IN_Reset OR TON_Watchdog.Q);
IF TrigReset.Q THEN
	FIFO.A_Reset();
	cmdStart := FALSE;
END_IF

TrigStart(CLK := CmdStart);
IF TrigStart.Q THEN
	ETAPE := 1;
END_IF


RsStart(SET := TrigStart.Q);
IF RsStart.Q1 THEN
	RequeteEntete :=  concat(concat(' INSERT INTO "',NomTable),'" ');
END_IF
		
CASE ETAPE OF
		
	1: // CONNECTED
		OUT_Busy := TRUE;
		IF SQLDatabase1.CreateCmd(pSQLCommand := ADR(SQLCommand1)) THEN 
			IF NOT SQLDatabase1.bError THEN
				MEMCPY(srcAddr:= ADR(RequeteEntete), destAddr := ADR(requeteFinale), n:= SIZEOF(RequeteEntete));
				pPosRequete := LEN(STR := RequeteEntete);
				Tmp_Nb_Buffer :=UDINT_TO_DINT(FIFO.nCount -1);
				FOR KK:= 1 TO MIN(Tmp_Nb_Buffer,CstNbLigneBuffer-1) DO
					fifo.A_Get();
					sTimeStamp	:=  ULINT_TO_STRING(fifo.Out.Timestamp);
					Format(sFormat := 'select $'%s$',%d,%5.2f FROM RDB$$DATABASE UNION ALL ', arg1 := F_STRING(sTimeStamp),arg2:= F_DINT(fifo.out.ParentId), arg3:= F_LREAL(fifo.out.Value), arg5:= F_STRING(NomTable), sOut=>sInsertValue);
					MEMCPY(srcAddr:= ADR(sInsertValue), destAddr := ADR(requeteFinale)+DINT_TO_DWORD(pPosRequete), n:= SIZEOF(sInsertValue));
					pPosRequete:= pPosRequete + LEN(STR := sInsertValue);
					fifo.A_Remove();
				END_FOR
				fifo.A_Get();
				sTimeStamp	:=  ULINT_TO_STRING(fifo.Out.Timestamp);
				Format(sFormat := 'select $'%s$',%d,%5.2f FROM RDB$$DATABASE;', arg1 := F_STRING(sTimeStamp),arg2:= F_DINT(fifo.out.ParentId), arg3:= F_LREAL(fifo.out.Value), sOut=>sInsertValue);
				MEMCPY(srcAddr:= ADR(sInsertValue), destAddr := ADR(requeteFinale)+DINT_TO_DWORD(pPosRequete), n:= SIZEOF(sInsertValue));
				fifo.A_Remove();
				IF Tmp_Nb_Buffer > 0 THEN
					ETAPE := 2;
				END_IF
			ELSIF SQLDatabase1.bError THEN
				ETAPE := 255;
			END_IF
		END_IF
	2:

		IF SQLCommand1.Execute(pSQLCmd := ADR(RequeteFinale), cbSQLCmd := SIZEOF(Requetefinale))THEN
			
			IF  NOT SQLCommand1.bError THEN
				ETAPE := 4;
			ELSIF SQLCommand1.bError THEN
				ETAPE := 255;
			END_IF
		END_IF

	4:
		IF NOT SQLDatabase1.bError THEN
			
			RequeteFinale := RequeteFinaleNull;
			
			//RequeteFinale := '';
			Tmp_Nb_Buffer := MIN(UDINT_TO_DINT(FIFO.nCount),CstNbLigneBuffer);
			//FOR KK:= 1 TO Tmp_Nb_Buffer DO
			//	fifo.A_Remove();
			//END_FOR
			TrigStart(CLK := FALSE);
			RsStart(RESET1 := TRUE);
			RsStart(RESET1 := FALSE);
			TrigCmdExec(CLK := FALSE);
			CmdStart := FALSE;
			Etape := 0;
			OUT_Error := FALSE;
			OUT_Busy := FALSE;

		ELSE 
			ETAPE := 255;
		END_IF
	255: 
		RequeteFinale := RequeteFinaleNull;

		SQLCommand1 := SQLCommand2;
		SQLDatabase1 := SQLDatabase2;
		OUT_Error := TRUE;
		RsStart(RESET1 := TRUE);
		RsStart(RESET1 := FALSE);
		TrigCmdExec(CLK := FALSE);
		CmdStart := FALSE;
		ETAPE := 0;
		OUT_Busy := FALSE;
END_CASE

METHOD M_AddLine : BOOL
VAR_INPUT
	InStruct			: St_DataHisto_Epoch;
END_VAR

VAR
END_VAR
fifo.in := InStruct;
fifo.A_Add();
END_METHOD

METHOD M_AlarmManager : BOOL
VAR_INPUT
	AlarmCode : WORD;
	
END_VAR


AlarmCode.0 := bBufferMaxFull;
AlarmCode.1 := bInStructNull;
END_METHOD

METHOD M_Connect : BOOL

VAR_OUTPUT
END_VAR
VAR_INPUT
	IN_hDBID				: DINT;
	IN_Start				: BOOL;
END_VAR
TrigStartConnect(CLK := IN_Start);
RsStartConnect(SET := TrigStartConnect.Q);
IF RsStartConnect.Q1 THEN
	IF SQLDatabase1.Connect(hDBID := IN_hDBID) THEN;
		RsStartConnect(RESET1 := TRUE);
		RsStartConnect(RESET1 := FALSE);
		bReconnect := FALSE;
	END_IF
END_IF

Out_Connected := SQLDatabase1.bConnected;
IF NOT OUT_Connected THEN
	btest := TRUE;
	
END_IF
END_METHOD

METHOD M_Disconnect : BOOL
VAR_INPUT
END_VAR
VAR_INPUT
	IN_Start				: BOOL;
END_VAR
TrigStartDisconnect(CLK := IN_Start);
RsStartDisconnect(SET := TrigStartDisconnect.Q);
IF RsStartDisconnect.Q1 THEN
	IF SQLDatabase1.Disconnect() THEN;
		RsStartDisconnect(RESET1 := TRUE);
		RsStartDisconnect(RESET1 := FALSE);
	END_IF
END_IF

Out_Connected := SQLDatabase1.bConnected;
END_METHOD

METHOD M_Init

VAR
	LL	: SINT;
	KK 	: SINT;
END_VAR
//Initialisation BUFFER
	//Buffer pour la lecture des sms
	FIFO.A_Reset();
	FIFO.A_Add();
	FIFO.A_Get();
	FIFO.A_Remove();
END_METHOD

END_FUNCTION_BLOCK

// ---- 00_FunctionsBlocks/Beckhoff/Database/Firebird/Firebird_ReadAlarms.TcPOU
PROGRAM Firebird_ReadAlarms
VAR_INPUT
	ParamTimeBetweenReconnect	: TIME := T#1M;
	IN_StartRead				: BOOL;
	IN_FrequencyRead			: TIME := T#1M;
	IN_bAct						: BOOL; // Read only Active values
	IN_FilterAct				: BOOL;
	IN_bAck						: BOOL; // Read only Acknowledged values
	IN_FilterAck				: BOOL;
	
	IN_TimeStampStart			: TIMESTRUCT;
	IN_TimeStampEnd				: TIMESTRUCT;
	
END_VAR
VAR CONSTANT
	NbMaxElements	 			: UINT := 250;
END_VAR
VAR_OUTPUT
	OUT_Busy					: BOOL;
	
END_VAR
VAR
	
	AX_Buffer_Alarms			: ARRAY[1..NbMaxElements] OF St_AlarmsV2;		// Buffer of alarms to write
	StNull						: St_AlarmsV2;		// Buffer of alarms to write
		
	// Connexion
		TP_Reconnect			: TP;
		Trig_Connect			: R_TRIG;
		TRIG_CmdStart			: R_TRIG;
		RS_Connect				: RS;
		RS_HasBeenConnected		: RS;
	// DISCONNECT
		TrigStartDisconnect				: R_TRIG;
		RsStartDisconnect				: RS;		
			
	// READ File       
		TP_ReadBddPeriodically	: TP;
		TRIG_ReadBddPeriodically: R_TRIG;

		ETAPE					: UINT;
		Trig_Start				: R_TRIG;   
		RS_Start				: RS; 	
		Requete					: ARRAY[1..10] OF STRING(1000);
		RequeteNull				: ARRAY[1..10] OF STRING(1000);
		sToAdd					: STRING(1000);
		pPosRequete				: DINT;
		TimeStampNull			: TIMESTRUCT;
		TimeStampDefault		: TIMESTRUCT;
		sTimeStampStart			: STRING(255);
		sTimeStampEnd			: STRING(255);
		sValue					: STRING(255);
		sAck					: STRING(255);
		Format					: FB_FormatString;
		SQLDatabase				: FB_SQLDatabaseEvt('',T#10S);
		SQLCommand				: FB_SQLCommandEvt('',T#10S);
		SQLCommandNull			: FB_SQLCommandEvt('',T#10S);
		SQLResult				: FB_SQLResultEvt('',T#10S);
		
	
	// General variables
		nbMax					: UINT;
		bInit 					: BOOL;
		NomTableAlarms			: STRING(255) := 'TABLE_ALARMS_V2';
		KK						: UINT;
		
	//TABLEAU
	
		AX_MesAlarmCode_Bool	: ARRAY [1..CstNbAlarmCode] OF ARRAY[1..15] OF BOOL; //Tableau de tous les alarmesCode en Bool
		AX_Alarm_State			: ARRAY [1..CstNbAlarmCode] OF ARRAY[1..15] OF BOOL; //Tableau de Bool avec toutes les nouveaux bit modifiés
		AX_MesAck				: ARRAY [1..CstNbAlarmCode] OF ARRAY[1..15] OF BOOL;
		AX_Ack_State			: ARRAY [1..CstNbAlarmCode] OF ARRAY[1..15] OF BOOL; //Tableau de Bool avec tous les nouveaux acknowledgement 

	

END_VAR

// DataProcessing
IF NOT bInit THEN
	M_Init();
END_IF
RS_HasBeenConnected(SET := SQLDatabase.bConnected);
TP_Reconnect(In :=RS_HasBeenConnected.Q1 AND NOT SQLDatabase.bConnected OR NOT bInit OR TP_Reconnect.Q, PT := ParamTimeBetweenReconnect);
	
TP_ReadBddPeriodically(IN := NOT TP_ReadBddPeriodically.Q, PT := IN_FrequencyRead);
TRIG_ReadBddPeriodically(CLK := TP_ReadBddPeriodically.Q);
TRIG_CmdStart(CLK := IN_StartRead);

Trig_Start(CLK := SQLDatabase.bConnected AND NOT OUT_Busy AND ( TRIG_CmdStart.Q OR TRIG_ReadBddPeriodically.Q));
IF Trig_Start.Q THEN
	// Init the table :
	FOR KK := 1 TO 10 DO 
		Requete[KK] := RequeteNull[KK];
	END_FOR
	FOR KK := 1 TO NbMaxElements DO
		AX_Buffer_Alarms[KK] := StNull;
	END_FOR
	Requete := RequeteNull;
	nbMax := NbMaxElements;
	pPosRequete := 0;
	// Je commence par préparer ma requête 
	IF MEMCMP(pBuf1 := ADR(IN_TimeStampStart), pBuf2:=ADR(TimeStampNull), n:=SIZEOF(TimeStampNull))=0 THEN
		IN_TimeStampStart := TimeStampDefault;
	END_IF
	sTimeStampStart := systemtime_to_string(in := IN_TimeStampStart);
	sTimeStampEnd := systemtime_to_string(in := IN_TimeStampEnd);
	Format( sFormat := 'Select first %d "TIMESTAMP_START", case when "TIMESTAMP_STOP" is null then cast($'01.01.1970, 00:00:00.000$' as timestamp) else "TIMESTAMP_STOP" end,AlarmsID,Act,Ack from %s where "TIMESTAMP_START" > $'%s$' ', 
		sOut=> sToAdd,
		arg1 := F_UINT(In:=nbMax),
		arg2 := F_STRING(In := NomTableAlarms),
		arg3 := F_STRING(in := sTimeStampStart)
	);
	MEMCPY(destAddr := ADR(requete), srcAddr := ADR(sToAdd), n := SIZEOF(sToAdd));
	pPosRequete:= pPosRequete + LEN(STR := sToAdd);
	
	IF IN_FilterAct THEN
		sToAdd := CONCAT(STR1 := ' AND Act = ', STR2 := UINT_TO_STRING(BOOL_TO_UINT(IN_bAct)));
		MEMCPY(srcAddr:= ADR(sToAdd), destAddr := ADR(Requete)+DINT_TO_DWORD(pPosRequete), n:= SIZEOF(sToAdd));
		pPosRequete:= pPosRequete + LEN(STR := sToAdd);
	END_IF
	
	IF IN_FilterAck THEN
		sToAdd := CONCAT(STR1 := ' AND Ack = ', STR2 := UINT_TO_STRING(BOOL_TO_UINT(IN_bAck)));
		MEMCPY(srcAddr:= ADR(sToAdd), destAddr := ADR(Requete)+DINT_TO_DWORD(pPosRequete), n:= SIZEOF(sToAdd));
		pPosRequete:= pPosRequete + LEN(STR := sToAdd);
	END_IF	

	sToAdd := ' order by TIMESTAMP_START desc';
	MEMCPY(srcAddr:= ADR(sToAdd), destAddr := ADR(Requete)+DINT_TO_DWORD(pPosRequete), n:= SIZEOF(sToAdd));
	pPosRequete:= pPosRequete + LEN(STR := sToAdd);	
	ETAPE := 1;
END_IF
		
CASE ETAPE OF
	1: // CONNECTED
		OUT_Busy := TRUE;
		IF SQLDatabase.CreateCmd(pSQLCommand := ADR(SQLCommand)) THEN 
			IF NOT SQLCommAND bError THEN
				ETAPE := 2;
			ELSIF SQLCommAND bError THEN
				ETAPE := 255;
			END_IF
		END_IF
		
	2:	
		IF SQLCommAND ExecuteDataReturn(pSQLCmd := ADR(Requete), cbSQLCmd := SIZEOF(Requete), pSQLDBResult := ADR(SQLResult))THEN
			IF  NOT SQLCommAND bError THEN
				ETAPE := 3;
			ELSIF SQLCommAND bError THEN
				ETAPE := 255;
			END_IF
		END_IF
	3: 
		IF SQLResult.Read(nStartIndex := 1, nRecordCount := NbMaxElements, pData := ADR(AX_Buffer_Alarms), cbData := SIZEOF(AX_Buffer_Alarms), bDataRelease := TRUE, bWithVerifying := FALSE) THEN
			IF NOT SQLResult.bError THEN
				Etape := 4;
			ELSE
				ETAPE := 255;
			END_IF
		END_IF
	4:
		IF NOT SQLDatabase.bError THEN

			Requete  := RequeteNull;
			Trig_Start(CLK := FALSE);
			Etape := 0;
			OUT_Busy := FALSE;
		ELSE 
			ETAPE := 255;
		END_IF
	255: 
		OUT_Busy := FALSE;
		Requete := RequeteNull;
		Etape := 0;
		IN_StartRead := FALSE;
END_CASE

METHOD M_Connect : BOOL

VAR_OUTPUT
END_VAR
VAR_INPUT
	IN_hDBID				: DINT;
	IN_Start				: BOOL;
END_VAR
Trig_Connect(CLK := IN_Start);
RS_Connect(SET := Trig_Connect.Q);
IF RS_Connect.Q1 THEN
	IF SQLDatabase.Connect(hDBID := IN_hDBID) THEN;
		RS_Connect(RESET1 := TRUE);
		RS_Connect(RESET1 := FALSE);
	END_IF
END_IF
END_METHOD

METHOD M_Disconnect : BOOL
VAR_INPUT
END_VAR
VAR_INPUT
	IN_Start				: BOOL;
END_VAR
TrigStartDisconnect(CLK := IN_Start);
RsStartDisconnect(SET := TrigStartDisconnect.Q);
IF RsStartDisconnect.Q1 THEN
	IF SQLDatabase.Disconnect() THEN;
		RsStartDisconnect(RESET1 := TRUE);
		RsStartDisconnect(RESET1 := FALSE);
	END_IF
END_IF
END_METHOD

METHOD M_Init

VAR
	LL	: SINT;
	KK 	: SINT;
END_VAR
TimeStampDefault.wYear := 1995;
TimeStampDefault.wMonth := 3;
TimeStampDefault.wDay := 12;

bInit := TRUE;
END_METHOD

END_PROGRAM

// ---- 00_FunctionsBlocks/Beckhoff/Database/Firebird/Firebird_RetrieveHDBID.TcPOU
PROGRAM Firebird_RetrieveHDBID
VAR_INPUT
	IN_ConfigDbActuelle		: ARRAY[0..MAX_CONFIGURATIONS] OF ST_ConfigDB; 
	IN_Dir					: T_MAXSTRING;
	IN_Name					: ARRAY[1..CstNbBases] OF STRING;
	IN_Start				: BOOL;
	IN_IpAddressServer		: STRING := 'localhost';
	IN_Port					: STRING := '3050';
END_VAR

VAR_OUTPUT
	OUT_hDBID         		: ARRAY[1..CstNbBases] OF DINT;	
	OUT_Error				: BOOL;
	OUT_Busy				: BOOL;
	OUT_Result				: INT;
END_VAR
VAR
	TrigStart				: R_TRIG;
	KK 						: UDINT;
	sExtension				: STRING;
	DbFullDirName			:  ARRAY[1..CstNbBases] OF STRING;
	LL						: DINT := 1;
	RS_Start				: RS;
END_VAR


sExtension := '.FDB';
FOR KK := 1 TO CstNbBases DO
	DbFullDirName[KK] := CONCAT(str1:= IN_IpAddressServer, STR2:= CONCAT(str1:= '/',str2:= CONCAT(STR1:= IN_Port, str2:=concat(str1 := ':', str2:=Concat(STR1:=Concat(STR1:= IN_Dir, STR2 := IN_Name[KK]), STR2 := sExtension)))));
END_FOR
TrigStart(CLK := IN_Start );
IF TrigStart.Q THEN
	LL := 1;
END_IF
RS_Start(SET := TrigStart.Q);
IF RS_Start.Q1 THEN

	OUT_Busy := TRUE;
	IF LL <= CstNbBases AND LL >0 THEN
		FOR KK := 0 TO MAX_CONFIGURATIONS DO
			IF IN_ConfigDbActuelle[KK].sDatabase = DbFullDirName[LL] THEN
				OUT_hDBID[LL] := IN_ConfigDbActuelle[KK].hDBID;
				LL := LL+1;
				EXIT;
			END_IF
			IF KK = MAX_CONFIGURATIONS THEN
				OUT_Result := -2;
				LL := -2;
				OUT_Error := TRUE;
				OUT_Busy := FALSE;
			END_IF
		END_FOR
	ELSIF LL > CstNbBases THEN
		OUT_Result := 1;
		OUT_Busy := FALSE;
		OUT_Error := FALSE;
		LL := 1;
		RS_Start(RESET1 := TRUE);
		RS_Start(RESET1 := FALSE);
	END_IF
END_IF

END_PROGRAM

// ---- 00_FunctionsBlocks/Beckhoff/Database/Firebird/Firebird_SelectBuffer.TcPOU
FUNCTION_BLOCK Firebird_SelectBuffer
VAR CONSTANT
	CstNbLigne							: DINT:= 250;
                            			
END_VAR                     			
                            			
VAR_INPUT                   			
	IN_NomTable							: STRING := 'Table100ms';
	IN_IdToSelect						: UINT;
	IN_TimeStampStart					: TIMESTRUCT;
	IN_hDBID							: UDINT;
	IN_Reset							: BOOL;
	IN_Start							: BOOL;
END_VAR  
VAR_OUTPUT                  			
	OUT_Error							: BOOL;
	OUT_Busy							: BOOL;
	OUT_Result							: INT;
	Out_Connected						: BOOL;
	Out_Array							: ARRAY[1..CstNbLigne] OF St_DataHisto;
END_VAR 

VAR                         			
	ETAPE								: UINT;
	NbLigne								: DINT;                        			
	TrigReset							: R_TRIG;
	
	StringTimeStart						: STRING;
		                    			
	StructNull							: St_DataHisto;
                            			
    SQLDatabase							: FB_SQLDatabaseEvt('',T#10S);
	SQLCommand							: FB_SQLCommandEvt('',T#10S);
	SQLCommandNull						: FB_SQLCommandEvt('',T#10S);
	SQLResult	 						: FB_SQLResultEvt(sNetID:='', tTimeout   := T#5S); 
	bConnected							: BOOL;              	        	
                            			
	pPosRequete							: DINT;                		
	RequeteFinale						: STRING(1000);	
	RequeteFinaleNull					: STRING(1000);	
	sTimeStamp							: STRING(255);  
	Format								: FB_FormatString;
	                			
	KK									: DINT;
	                    				
	CmdStart							: BOOL;
	TrigCmdExec							: R_TRIG;
	TrigStart							: R_TRIG;
	RsStart								: RS;
	                        			
	// AlarmManagement      			
		bBufferMaxFull 					: BOOL;        		
		bInStructNull					: BOOL;
		
	// CONNECT	
		TrigStartConnect				: R_TRIG;	
		RsStartConnect					: RS;
END_VAR

TrigReset(CLK := IN_Reset);
IF TrigReset.Q THEN

	//SQLCommand := SQLCommandNull;
END_IF

TrigStart(CLK := IN_Start);
IF TrigStart.Q THEN
	NbLigne := CstNbLigne;
	StringTimeStart := LEFT(STR := SYSTEMTIME_TO_STRING(IN_TimeStampStart), SIZE := LEN(SYSTEMTIME_TO_STRING(IN_TimeStampStart))-4);
	
	Format(sFormat := 'Select first %d * from "%s" where "ParentId" = %d and "TimeStamp" > $'%s$'', sOut => RequeteFinale, 
	arg1 := F_DINT(in := NbLigne), arg2 := F_STRING(in := IN_NomTable), arg3 := F_UINT(in := IN_IdToSelect), arg4:= F_STRING(in := StringTimeStart));
	ETAPE := 1;
END_IF

CASE ETAPE OF
		
	1: // CONNECTED
		IF SQLDatabase.CreateCmd(pSQLCommand := ADR(SQLCommand)) THEN 
			IF NOT SQLCommAND bError THEN
				ETAPE := 2;
			ELSIF SQLCommAND bError THEN
				ETAPE := 255;
			END_IF
		END_IF
	2:
		
		IF SQLCommAND ExecuteDataReturn(pSQLCmd := ADR(RequeteFinale), cbSQLCmd := SIZEOF(RequeteFinale), pSQLDBResult := ADR(SQLResult)) THEN
    		IF SQLCommAND bError THEN
    		    ETAPE := 255; 
    		ELSE
    		    ETAPE := 3; 
    		END_IF			
		END_IF
	3:
		IF SQLResult.Read(nStartIndex := 0, nRecordCount := CstNbLigne, pData := ADR(Out_Array), cbData := SIZEOF(Out_Array), bWithVerifying := TRUE, bDataRelease:= TRUE) THEN
			IF NOT SQLResult.bError THEN
				ETAPE := 4;
			ELSE
				ETAPE := 255;
			END_IF
		END_IF
		
	4:
		IF NOT SQLDatabase.bError THEN
			
			RequeteFinale := RequeteFinaleNull;
	
			TrigStart(CLK := FALSE);
			RsStart(RESET1 := TRUE);
			RsStart(RESET1 := FALSE);
			TrigCmdExec(CLK := FALSE);
			IN_Start := FALSE;
			Etape := 0;
			OUT_Error := FALSE;
		ELSE 
			ETAPE := 255;
		END_IF
	255: 
		RequeteFinale := RequeteFinaleNull;
		//RequeteFinale := '';
		OUT_Error := TRUE;
		Etape := 0;
		RsStart(RESET1 := TRUE);
		RsStart(RESET1 := FALSE);
		TrigCmdExec(CLK := FALSE);
		IN_Start := FALSE;
END_CASE

METHOD M_Connect : BOOL

VAR_OUTPUT
END_VAR
VAR_INPUT
	IN_hDBID				: UDINT;
	IN_Start				: BOOL;
END_VAR
TrigStartConnect(CLK := IN_Start);
RsStartConnect(SET := TrigStartConnect.Q);
IF RsStartConnect.Q1 THEN
	IF SQLDatabase.Connect(hDBID := IN_hDBID) THEN;
		RsStartConnect(RESET1 := TRUE);
		RsStartConnect(RESET1 := FALSE);
	END_IF
END_IF

Out_Connected := SQLDatabase.bConnected;
END_METHOD

END_FUNCTION_BLOCK

// ---- 00_FunctionsBlocks/Beckhoff/Database/Firebird/Firebird_WriteAlarms.TcPOU
PROGRAM Firebird_WriteAlarms
VAR_INPUT
	ParamTimeBetweenReconnect	: TIME := T#1M;
	IN_Reset					: BOOL;
	
	FIFO						: FB_DBDatasetFifo;
END_VAR
VAR_OUTPUT
END_VAR
	
VAR

	CmdStart					: BOOL;
	CmdReset					: BOOL;
	// Data processing 
	MesDataExd			: LoggerFirebird ; 
	// RESET
		Trig_Reset				: R_TRIG;
		
	// Connexion
		TP_Reconnect			: TP;
		Trig_Connect			: R_TRIG;
		RS_Connect				: RS;
		RS_HasBeenConnected		: RS;
	// DISCONNECT
		TrigStartDisconnect				: R_TRIG;
		RsStartDisconnect				: RS;		
		
		
	// Write File       
		ETAPE					: UINT;
		Trig_Start				: R_TRIG;   
		Requete					: STRING(1000);
		sTimeStamp 				: STRING(255);
		sTimeStamp_Ms			: STRING(255);
		sValue					: STRING(255);
		sAck					: STRING(255);
		Format					: FB_FormatString;
		SQLDatabase				: FB_SQLDatabaseEvt('',T#10S);
		SQLCommand1				: FB_SQLCommandEvt('',T#10S);
		SQLCommandNull			: FB_SQLCommandEvt('',T#10S);
		
	
	// General variables
		bInit 					: BOOL;

		NomTable				: STRING(255) := 'TABLE_ALARMS';
		

	
END_VAR

// DataProcessing
IF NOT bInit THEN
	M_Init();
END_IF
RS_HasBeenConnected(SET := SQLDatabase.bConnected);
TP_Reconnect(In :=RS_HasBeenConnected.Q1 AND NOT SQLDatabase.bConnected OR NOT bInit OR TP_Reconnect.Q, PT := ParamTimeBetweenReconnect);
	
M_AlarmManager();


Trig_Reset(CLK := IN_Reset OR CmdClearFault_G);
IF Trig_Reset.Q THEN
	FIFO.A_Reset();
	SQLCommand1 := SQLCommandNull;
	CmdReset := False;
END_IF


// La première ligne est non nulle
CmdStart := FIFO.nCount >0 AND SQLDatabase.bConnected;
Trig_Start(CLK := CmdStart);
IF Trig_Start.Q THEN
	ETAPE := 1;
END_IF
		
CASE ETAPE OF
	1: // CONNECTED
		IF SQLDatabase.CreateCmd(pSQLCommand := ADR(SQLCommand1)) THEN 
			IF NOT SQLCommand1.bError THEN
				ETAPE := 2;
			ELSIF SQLCommand1.bError THEN
				ETAPE := 255;
			END_IF
		END_IF
		
	2:
		//sTimeStamp := left(STR := (AX_Buffer_Alarms[1].TimeStamp_Act), SIZE := LEN((AX_Buffer_Alarms[1].TimeStamp_Act))-4);
		FIFO.A_Get();	
		sTimeStamp := FIFO.OUT.TimeStamp_Act;
		sTimeStamp_MS := right(STR := (sTimeStamp), SIZE := 3);	
		sValue	:= INT_TO_STRING(BOOL_TO_INT(FIFO.Out.Value));
		sAck	:= INT_TO_STRING(BOOL_TO_INT(FIFO.Out.Ack));
		Format(sFormat := 'Insert into %s values ( $'%s$',%d, %s, %s);', 
			sOut => Requete,
			arg1 := F_STRING(in := NomTable),
			arg2 := F_STRING(in := sTimeStamp),
			arg3 := F_UINT(in := FIFO.Out.ID),
			arg4 := F_STRING(in := sValue),
			arg5 := F_STRING(in := sAck)
		);
		IF SQLCommand1.Execute(pSQLCmd := ADR(Requete), cbSQLCmd := SIZEOF(Requete))THEN
			IF  NOT SQLCommand1.bError THEN
				ETAPE := 4;
			ELSIF SQLCommand1.bError THEN
				ETAPE := 255;
			END_IF
		END_IF

	4:
		IF NOT SQLDatabase.bError THEN
			FIFO.A_Remove();
			Requete  := '';
			Trig_Start(CLK := FALSE);
			Etape := 0;
		ELSE 
			ETAPE := 255;
		END_IF
		
	255: 
		CmdReset := TRUE;
		Requete := '';
		Etape := 0;
		CmdStart := FALSE;
END_CASE

METHOD M_AlarmManager
VAR
	FB_AlarmCodeManager : FB_AlarmCodeManager;
END_VAR
// Gestion des alarmes internes au code

FB_AlarmCodeManager
(
	bAlarm1 := SQLCommand1.bError,				// Insert new alarm failed
	bAlarm2 := SQLDatabase.bError,				// Connexion to database failed
	bAlarm3 := FALSE,							// 
	bAlarm4 := FIFO.bOverwrite,					// Fifo Overflow
	bAlarm5 :=FALSE,							//
	bAlarm6 :=FALSE,    						//
	bAlarm7 :=FALSE,    						//
	bAlarm8 :=FALSE,    						//
	bAlarm9 :=FALSE,    						//
	bAlarm10 :=FALSE,   						//
	bAlarm11 :=FALSE,   						//
	bAlarm12 :=FALSE,   						//
	bAlarm13 :=FALSE,   						//
	bAlarm14 :=FALSE,   						//
	bAlarm15 :=FALSE,							//	
	
	wAlarmCode =>MesDataExd.MesData.MesAlarmCode
);
END_METHOD

METHOD M_Connect : BOOL

VAR_OUTPUT
END_VAR
VAR_INPUT
	IN_hDBID				: DINT;
	IN_Start				: BOOL;
END_VAR
Trig_Connect(CLK := IN_Start);
RS_Connect(SET := Trig_Connect.Q);
IF RS_Connect.Q1 THEN
	IF SQLDatabase.Connect(hDBID := IN_hDBID) THEN;
		RS_Connect(RESET1 := TRUE);
		RS_Connect(RESET1 := FALSE);
	END_IF
END_IF
END_METHOD

METHOD M_Disconnect : BOOL
VAR_INPUT
END_VAR
VAR_INPUT
	IN_Start				: BOOL;
END_VAR
VAR
END_VAR
TrigStartDisconnect(CLK := IN_Start);
RsStartDisconnect(SET := TrigStartDisconnect.Q);
IF RsStartDisconnect.Q1 THEN
	IF SQLDatabase.Disconnect() THEN;
		RsStartDisconnect(RESET1 := TRUE);
		RsStartDisconnect(RESET1 := FALSE);
	END_IF
END_IF
END_METHOD

METHOD M_Init

VAR
	LL	: SINT;
	KK 	: SINT;
END_VAR
//Initialisation BUFFER
	//Buffer pour la lecture des sms
	FIFO.A_Reset();
	FIFO.A_Add();
	FIFO.A_Get();
	FIFO.A_Remove();
	
	FIFO.In.Message :=  'Activation du code';
	FIFO.In.TimeStamp_Act := SYSTEMTIME_TO_STRING(CalLocalTimeStruct); 
	FIFO.A_Add();
	bInit := TRUE;
END_METHOD

END_PROGRAM

// ---- 00_FunctionsBlocks/Beckhoff/Database/InfluxDb/InfluxDb_ReadValues.TcPOU
PROGRAM InfluxDb_ReadValues
               					
VAR_INPUT  
	IN_TimeStart							: LINT;
	IN_bRead								: BOOL;             					
	IN_Dbid									: UINT := 1;
	IN_NbRecordRead							: UINT := 100;
	IN_bAck									: BOOL;	// Filter value for acknowledged filter
	IN_bVal									: BOOL; // Filter value for value filter
	IN_FilterAck							: BOOL; // Is the acknowledged filter active 
	IN_FilterVal							: BOOL; // Is the value filter active 
	IN_Database								: T_MaxString;
END_VAR

VAR_OUTPUT
    OUT_bError								: BOOL;
	OUT_bBusy								: BOOL;
	OUT_pTableResults						: PVOID;
	OUT_cbTableResults						: UINT;
END_VAR

VAR
	Query									: T_MaxString;
	QueryInit								: T_MaxString := 'SELECT time, Message, ID, Value, Ack  FROM %s.autogen.Alarms  ';
	QueryOrder								: T_MaxString := ' order by time desc limit %d';
	QueryFinal								: T_MaxString ;
	
    QueryOption_TSDB_Select 				: T_QueryOptionTimeSeriesDB_Query; 
    fbNoSQLQueryBuilder_TimeSeriesDB 		: FB_NoSQLQueryBuilder_TimeSeriesDB; 
    fbNoSqlQueryEvt 						: FB_NoSQLQueryEvt(sNetID := '', tTimeout := T#15S); 
	fbNoSqlResultEvt						: FB_NoSQLResultEvt(sNetID := '', tTimeout := T#15S);
	fbNoSqlValidationEvt					: FB_NoSQLValidationEvt(sNetID := '', tTimeout := T#15S);
	nState 									: UINT;
	ReaDS_Transfouct								: ARRAY[1..250]OF ST_InfluxAlarmsRetrieve;
	Format									: FB_FormatString;          						

END_VAR

fbNoSQLQueryBuilder_TimeSeriesDB.pQueryOptions := ADR(QueryOption_TSDB_Select);
fbNoSQLQueryBuilder_TimeSeriesDB.cbQueryOptions := SIZEOF(QueryOption_TSDB_Select);

OUT_pTableResults 	:= ADR(ReaDS_Transfouct);
OUT_cbTableResults 	:= SIZEOF(ReaDS_Transfouct);

IF IN_bRead THEN
	OUT_bBusy 	:= TRUE;
	IN_bRead 	:= FALSE;
	nState 		:= 1;
	Query := QueryInit;
	IF IN_FilterAck OR IN_FilterVal THEN
		query := concat(STR1 := query, str2 := 'Where ');
		
		IF IN_FilterAck THEN
			query := concat(STR1:= query, STR2 := concat(STR1 := ' Ack=', str2 := BOOL_TO_STRING(IN_bAck)));
		END_IF
		
		IF IN_FilterAck AND IN_FilterVal THEN
			query := concat(STR1:= query, STR2 := ' AND ');
		END_IF
		
		IF IN_FilterVal THEN
			query := concat(STR1:= query, STR2 := concat(STR1 := 'Value=', str2 := BOOL_TO_STRING(IN_bVal)));
		END_IF
		
	END_IF
	query := concat(str1 := query, STR2 := QueryOrder);
	Format(sFormat := Query, arg1 := F_STRING(in:=IN_Database), arg2:= F_UINT(in:=IN_NbRecordRead), sOut => QueryFinal);
	
	QueryOption_TSDB_Select.cbQuery := SIZEOF(QueryFinal);
	QueryOption_TSDB_Select.pQuery := ADR(QueryFinal);
END_IF

CASE nState OF 
	1:
		IF fbNoSqlQueryEvt.ExecuteDataReturn(hDBID := IN_Dbid, iNoSQLQueryBuilder := fbNoSQLQueryBuilder_TimeSeriesDB, pNoSQLResult := ADR(fbNoSqlResultEvt)) THEN
			IF fbNoSqlQueryEvt.bError THEN
				OUT_bError := TRUE;
				nState := 0;
			ELSE
				nState := 2;
			END_IF
		END_IF
	2:
		IF fbNoSqlResultEvt.ReadAsStruct
		(
			nStartIndex := 0, 
			nRecordCount:= IN_NbRecordRead,  
			pData:= ADR(ReaDS_Transfouct),  
			cbData:= SIZEOF(ReaDS_Transfouct),  
			bValidate := TRUE,  
			bDataRelease:= TRUE,  
			pNoSQLValidation:= ADR(fbNoSqlValidationEvt) 
		) THEN
			IF fbNoSqlResultEvt.bError THEN
				OUT_bError := TRUE;
				OUT_bBusy := FALSE;
				nState := 0;
			ELSE
				nState := 3;
				OUT_bBusy := FALSE;
			END_IF
		END_IF
	
END_CASE

END_PROGRAM

// ---- 00_FunctionsBlocks/Beckhoff/Database/InfluxDb/InfluxDb_WriteAlarms.TcPOU
PROGRAM InfluxDb_WriteAlarms

VAR_INPUT
	IN_Dbid										: UINT;
	IN_FIFO										: FB_DBDatasetFifo_Influx;
	IN_Reset									: BOOL;
MesDataExd								: LoggerInfluxDb;
END_VAR

VAR
	// M_Init
		TP_Init									: TP;
		F_TRIG_Init								: F_TRIG;
   		bInit 									: BOOL;
	// Reset                					
		Trig_Reset								: R_TRIG;
	// Insert value             				
		CmdStart								: BOOL;
    	QueryOption_TSDB_Insert 				: T_QueryOptionTimeSeriesDB_Insert; // defines detailed Queryparameter
    	fbNoSQLQueryBuilder_TimeSeriesDB 		: FB_NoSQLQueryBuilder_TimeSeriesDB; // defines database type specific api
    	fbNoSqlQueryEvt 						: FB_NoSQLQueryEvt(sNetID := '', tTimeout := T#15S); // functionblock to execute queries
		nState 									: UINT;
		ValueToInsert							: ST_InfluxAlarmsInsert;
    // error handling helper values
    sErrorMessage								: STRING(255);

	
END_VAR

IF NOT bInit THEN
	M_Init();
END_IF

Trig_Reset(CLK := IN_Reset OR CmdClearFault_G);
IF Trig_Reset.Q THEN
	IN_Reset := FALSE;
	IN_FIFO.A_Reset();
END_IF

CmdStart := IN_FIFO.nCount >0 ;
IF CmdStart THEN
	CmdStart := FALSE;
	
	fbNoSQLQueryBuilder_TimeSeriesDB.pQueryOptions := ADR(QueryOption_TSDB_Insert);
	fbNoSQLQueryBuilder_TimeSeriesDB.cbQueryOptions := SIZEOF(QueryOption_TSDB_Insert);
	IN_FIFO.A_Get();
	ValueToInsert	:= IN_FIFO.Out;
	QueryOption_TSDB_Insert.sTableName 			:= 'Alarms';			
	QueryOption_TSDB_Insert.sDataType 			:= 'ST_InfluxAlarmsInsert';	
	QueryOption_TSDB_Insert.pSymbol 			:= ADR(ValueToInsert); 	
	QueryOption_TSDB_Insert.cbSymbol 			:= SIZEOF(ValueToInsert); 
	QueryOption_TSDB_Insert.nDataCount 			:= 1;					
	QueryOption_TSDB_Insert.nStartTimestamp 	:= F_GetSystemTime(); 	

	nState := 3;
END_IF

CASE nState OF 
    3:
        IF fbNoSqlQueryEvt.Execute(IN_Dbid, fbNoSQLQueryBuilder_TimeSeriesDB) THEN
			IF fbNoSqlQueryEvt.bError THEN
			MesDataExd.MesData.MesAlarmCode.1 := TRUE;
				nState := 1;
			ELSE
			MesDataExd.MesData.MesAlarmCode.1 := FALSE;
			   	nState := 1;
 				IN_FIFO.A_Remove();
           END_IF
        END_IF
END_CASE

METHOD M_Init : BOOL
VAR_INPUT
END_VAR
//Initialisation BUFFER
	//Buffer pour la lecture des sms
	IN_FIFO.A_Reset();
	IN_FIFO.A_Add();
	IN_FIFO.A_Get();
	IN_FIFO.A_Remove();
	
	IN_FIFO.In.Message :=  'Activation du code';
	IN_FIFO.A_Add();
	bInit := TRUE;
END_METHOD

END_PROGRAM

// ---- 00_FunctionsBlocks/Beckhoff/Database/InfluxDb/InfluxDb_WriteStruct.TcPOU
FUNCTION_BLOCK InfluxDb_WriteStruct
VAR_INPUT PERSISTENT
	ParamInitTime							: TIME := T#1S;
END_VAR                 					
VAR_INPUT               					
	IN_Table 								: STRING;
	IN_StructureName 						: STRING;
	IN_DataAddr								: PVOID;
	IN_DataSize								: UDINT;
	IN_NumberStructure						: UDINT;		// ArrayLength
	IN_DataFrequency						: TIME;
	IN_Dbid									: UINT;
END_VAR

VAR
    QueryOption_TSDB_Insert 				: T_QueryOptionTimeSeriesDB_Insert; // defines detailed Queryparameter
    fbNoSQLQueryBuilder_TimeSeriesDB 		: FB_NoSQLQueryBuilder_TimeSeriesDB; // defines database type specific api
    fbNoSqlQueryEvt 						: FB_NoSQLQueryEvt(sNetID := '', tTimeout := T#15S); // functionblock to execute queries
    bInit 									: BOOL;
	nState 									: UINT;
    Name 									: STRING;
	Current_Time 							: TIME;
	Old_Time	 							: TIME;
	
    // error handling helper values
    bError									: BOOL;
    sErrorMessage							: STRING(255);
                    						
	// InitWait     						
	TP_Init									: TP;
	F_TRIG_Init								: F_TRIG;
	
END_VAR

fbNoSQLQueryBuilder_TimeSeriesDB.pQueryOptions := ADR(QueryOption_TSDB_Insert);
fbNoSQLQueryBuilder_TimeSeriesDB.cbQueryOptions := SIZEOF(QueryOption_TSDB_Insert);

QueryOption_TSDB_Insert.sTableName 			:= IN_Table;			//'PcsTable1';
QueryOption_TSDB_Insert.sDataType 			:= IN_StructureName;	//'ST_Pcs';
QueryOption_TSDB_Insert.pSymbol 			:= IN_DataAddr; 		//ADR(AX_InvData);
QueryOption_TSDB_Insert.cbSymbol 			:= IN_DataSize; 		//SIZEOF(AX_InvData);
QueryOption_TSDB_Insert.nDataCount 			:= IN_NumberStructure;	//CstNbInv*CstNbPcs_Inv; 
QueryOption_TSDB_Insert.nStartTimestamp 	:= F_GetSystemTime(); 	// get current twincat time 
QueryOption_TSDB_Insert.nCycleTime		 	:= 0; 					// 0 : insert all structures at the same time

TP_Init(IN := NOT bInit OR CmdInit_G, PT := ParamInitTime);
F_TRIG_Init(CLK := TP_Init.Q);
IF F_TRIG_Init.Q THEN
	nState := 1;
END_IF


CASE nState OF 
    1: // init 
		Current_Time := TIME();
		IF Current_Time > Old_Time + IN_DataFrequency - INT_TO_TIME(CstCycleTime_G) THEN
			nState := 3;
			
		END_IF
    3: // write values 
		Old_Time := TIME();
        IF fbNoSqlQueryEvt.Execute(IN_Dbid, fbNoSQLQueryBuilder_TimeSeriesDB) THEN
            IF fbNoSqlQueryEvt.bError THEN
               bError := TRUE;
			   nState := 1;
            ELSE
				bError := FALSE;
			   	nState := 1;
            END_IF
        END_IF
	
END_CASE

END_FUNCTION_BLOCK

// ---- 00_FunctionsBlocks/Beckhoff/Database/PRG_EpochConverter.TcPOU
PROGRAM PRG_EpochConverter
//Convert Epoch to TimeStruct
VAR
	FileTime				: T_FILETIME;
	ConvertTime				: FB_SystemTimeToTzSpecificLocalTime;
END_VAR
VAR_INPUT
	IN_bIsWeird 			: BOOL; 				// Cas pour l'Epoch venant de Influx : offset de   82 011 087 
	IN_OffSet				: DINT :=  -82011087 ; 	// Cas pour l'Epoch venant de Influx : valeur de l'offset
	IN_Epoch				: LINT;					// Input 
END_VAR             		
VAR_OUTPUT          		
	OUT_TimeStruct_UTC		: TIMESTRUCT;
	OUT_TimeStruct_Local	: TIMESTRUCT;
END_VAR

IF IN_bIsWeird THEN
	IN_Epoch := IN_Epoch + IN_OffSet;
END_IF

FileTime.dwHighDateTime := LINT_TO_DWORD(SHR(IN_Epoch, 32));
FileTime.dwLowDateTime 	:= LINT_TO_DWORD(IN_Epoch);
OUT_TimeStruct_UTC 		:= FILETIME_TO_SYSTEMTIME( FileTime );
ConvertTime(in := OUT_TimeStruct_UTC, tzInfo := CstTimeZone_G, out => OUT_TimeStruct_Local);

END_PROGRAM

// ---- 00_FunctionsBlocks/Beckhoff/Database/PRG_TimestructConverter.TcPOU
PROGRAM PRG_TimestructConverter
//Convert TimeStruct to Epoch 
VAR
	DT_Time			: DT;
	FileTime		: T_FILETIME;
END_VAR
VAR_INPUT
	IN_TimeStruct			: TIMESTRUCT;					// Input 
END_VAR             		
VAR_OUTPUT          		
	OUT_Epoch		: LINT;
END_VAR

DT_Time 		:= SYSTEMTIME_TO_DT( IN_TimeStruct );

FileTime 		:= DT_TO_FILETIME(dtIn := DT_Time);

OUT_Epoch := (SHL(DWORD_TO_ULINT(FileTime.dwHighDateTime), 32) + DWORD_TO_ULINT(FileTime.dwLowDateTime)) / 10000000 - 11644473600;

END_PROGRAM

// ---- 00_FunctionsBlocks/Beckhoff/Database/SQLCe/FB_SQLExpert_InsertBuffer_1.TcPOU
FUNCTION_BLOCK FB_SQLExpert_InsertBuffer_1
// Fonctionnement : Tableau de 2000 structures en input. Dès qu'on atteint 1000 structures remplies, décalage de l'espace mémoire
// pour en 1 temps de cycle pour ne pas perdre de données sur le transfert.
VAR CONSTANT
	CstNbLigneBuffer		: DINT:= 500;
	CstNbLigneBufferMax	 	: DINT:= 5000;

END_VAR

VAR_INPUT
	NomTable				: STRING := 'Table100ms';
	hDBID					: UDINT;
END_VAR

VAR_OUTPUT
	OUT_Error				: BOOL;
	OUT_Busy				: BOOL;
END_VAR

VAR
	ETAPE					: UINT;

    myStruct      			: ARRAY[1..CstNbLigneBuffer] OF St_DataHisto;
	myStructMax    			: ARRAY[1..CstNbLigneBufferMax] OF St_DataHisto;
	StructNull				: St_DataHisto;

    SQLDatabase				: FB_SQLDatabaseEvt('',T#10S);
	SQLCommand1				: FB_SQLCommandEvt('',T#10S);
	SQLCommandNull			: FB_SQLCommandEvt('',T#10S);
	bConnected				: BOOL;              	        	

	TrameValues				: T_MaxString := ' ([Timestamp],[Timestamp_Ms],[ParentId],[Value])';
	pPosRequete				: DINT;                		
	RequeteFinale			: ARRAY[1..100] OF STRING(1000);	
	RequeteFinaleNull		: ARRAY[1..100] OF STRING(1000);	
	sTimeStamp				: STRING(255);               	
	RequeteEntete			: STRING(1000);
	sInsertValue			: STRING(1000);
	Format					: FB_FormatString;
	                		
	NbElemBuffer			: DINT;
	KK						: DINT;
	                    	
	CmdStart				: BOOL;
	TrigCmdExec				: R_TRIG;
	TrigStart				: R_TRIG;
	RsStart					: RS;
	
	// Insert
		hDBID_BaseTampon	: UINT := 3;
	// AlarmManagement      
		bBufferMaxFull 		: BOOL;        		
		bInStructNull		: BOOL;
		
		
		
	
END_VAR

NbElemBuffer := M_Count();
CmdStart := NbElemBuffer>= CstNbLigneBuffer;


TrigStart(CLK := CmdStart);
IF TrigStart.Q THEN
	FOR KK := 1 TO CstNbLigneBuffer DO
		myStruct[KK] := myStructMax[KK];
	END_FOR
END_IF


// call functionblock

CASE ETAPE OF
	0://INITIALISATION  & CONNECTION
		RequeteEntete := concat(concat('INSERT INTO ',NomTable),concat(TrameValues,' VALUES '));
		RsStart(SET := TrigStart.Q);
		IF RsStart.Q1 THEN
			IF SQLDatabase.Connect(hDBID := hDBID) THEN;
				bConnected := NOT sqldatabase.bError;
				IF bConnected THEN
					ETAPE := 1;
				ELSE
					ETAPE := 255;
				END_IF
			END_IF
		END_IF
		
	1: // CONNECTED
		IF SQLDatabase.CreateCmd(pSQLCommand := ADR(SQLCommand1)) THEN 
			IF NOT SQLCommand1.bError THEN
				ETAPE := 2;
			ELSIF SQLCommand1.bError THEN
				ETAPE := 255;
			END_IF
		END_IF
	2:
		MEMCPY(srcAddr:= ADR(RequeteEntete), destAddr := ADR(requeteFinale), n:= SIZEOF(RequeteEntete));
		pPosRequete := LEN(STR := RequeteEntete);
		FOR KK:= 1 TO CstNbLigneBuffer-1 DO
			sTimeStamp	:= right(STR := DT_TO_STRING(myStruct[KK].Timestamp), SIZE := LEN(DT_TO_STRING(myStruct[KK].Timestamp))-3);
			Format(sFormat := '($'%s $',%.3d,%.4d,%5.2f),', arg1 := F_STRING(sTimeStamp),arg2:=F_DINT(myStruct[KK].Timestamp_Ms), arg3:= F_DINT(myStruct[KK].ParentId), arg4:= F_LREAL(myStruct[KK].Value), sOut=>sInsertValue);
			MEMCPY(srcAddr:= ADR(sInsertValue), destAddr := ADR(requeteFinale)+DINT_TO_DWORD(pPosRequete), n:= SIZEOF(sInsertValue));
			pPosRequete:= pPosRequete + LEN(STR := sInsertValue);
		END_FOR
		sTimeStamp	:= right(STR := DT_TO_STRING(myStruct[KK].Timestamp), SIZE := LEN(DT_TO_STRING(myStruct[KK].Timestamp))-3);
		Format(sFormat := '($'%s $',%.3d,%.4d,%5.2f)', arg1 := F_STRING(sTimeStamp),arg2:=F_DINT(myStruct[KK].Timestamp_Ms), arg3:= F_DINT(myStruct[KK].ParentId), arg4:= F_LREAL(myStruct[KK].Value), sOut=>sInsertValue);
		MEMCPY(srcAddr:= ADR(sInsertValue), destAddr := ADR(requeteFinale)+DINT_TO_DWORD(pPosRequete), n:= SIZEOF(sInsertValue));
	
		IF SQLCommand1.Execute(pSQLCmd := ADR(RequeteFinale), cbSQLCmd := SIZEOF(Requetefinale))THEN
			
			IF  NOT SQLCommand1.bError THEN
				ETAPE := 3;
			ELSIF SQLCommand1.bError THEN
				ETAPE := 255;
			END_IF
		END_IF
	3:
			IF SQLDatabase.Disconnect() THEN
				ETAPE := 4;
			END_IF 
	4:
		IF NOT SQLDatabase.bError THEN
			RequeteFinale := RequeteFinaleNull;
			FOR KK := CstNbLigneBuffer TO CstNbLigneBufferMax -1 DO
				myStructMax[KK+1-CstNbLigneBuffer]:= myStructMax[KK+1];
			END_FOR
			
			FOR KK := CstNbLigneBufferMax-CstNbLigneBuffer+1 TO CstNbLigneBufferMax DO
				myStructMax[KK]:= StructNull;
			END_FOR			
			
			TrigStart(CLK := FALSE);
			RsStart(RESET1 := TRUE);
			RsStart(RESET1 := FALSE);
			TrigCmdExec(CLK := FALSE);
			CmdStart := FALSE;
			Etape := 0;
			OUT_Error := FALSE;
		ELSE 
			ETAPE := 255;
		END_IF
	255: 
		RequeteFinale := RequeteFinaleNull;
		OUT_Error := TRUE;
		Etape := 0;
		RsStart(RESET1 := TRUE);
		RsStart(RESET1 := FALSE);
		TrigCmdExec(CLK := FALSE);
		CmdStart := FALSE;
		
END_CASE

METHOD M_AddLine : BOOL
VAR_INPUT
	InStruct			: St_DataHisto;
END_VAR

VAR
END_VAR
// Check the biggest buffer isn't full
IF MEMCMP(pBuf1 := ADR(StructNull), pBuf2 := ADR(myStructMax[CstNbLigneBufferMax]), n := SIZEOF(StructNull)) <> 0 THEN
	bBufferMaxFull := TRUE;
ELSE
	//Check the input struct isn't null
	IF MEMCMP(pBuf1 := ADR(StructNull), pBuf2 := ADR(InStruct), n := SIZEOF(StructNull)) = 0 THEN
		bInStructNull := TRUE;
	ELSE
		// We parse the biggest buffer
		FOR KK := 1 TO CstNbLigneBufferMax DO 
			IF MEMCMP(pBuf1 := ADR(StructNull), pBuf2 := ADR(myStructMax[KK]), n := SIZEOF(StructNull)) = 0 THEN
				myStructMax[KK] := InStruct;
				bBufferMaxFull := FALSE;
				EXIT;
			END_IF
		END_FOR
	END_IF
END_IF
END_METHOD

METHOD M_AlarmManager : BOOL
VAR_INPUT
	AlarmCode : WORD;
	
END_VAR


AlarmCode.0 := bBufferMaxFull;
AlarmCode.1 := bInStructNull;
END_METHOD

METHOD M_Count : DINT
VAR_INPUT
END_VAR
VAR

END_VAR
FOR KK := 1 TO CstNbLigneBufferMax DO 

	IF MEMCMP(pBuf1 := ADR(StructNull), pBuf2 := ADR(myStructMax[KK]), n := SIZEOF(StructNull)) = 0 THEN
		EXIT ;
	END_IF
END_FOR

M_Count := MIN(KK, CstNbLigneBufferMax);
END_METHOD

END_FUNCTION_BLOCK

// ---- 00_FunctionsBlocks/Beckhoff/Database/SQLite/SQLite_CreateDb_V2_1.TcPOU
PROGRAM SQLite_CreateDb_V2_1
VAR_INPUT
	IN_ConfigDbActuelle		: ARRAY[0..MAX_CONFIGURATIONS] OF ST_ConfigDB; 
	IN_DbType				: UINT:= 1; // 1:T_DBConfig_SQLite, 2:T_DBConfig_SQLCe
	IN_Dir					: T_MAXSTRING;
	IN_Name					: STRING;
	IN_Start				: BOOL;
	IN_TableName			: STRING;
END_VAR
VAR_IN_OUT
	IN_hDBID         		: UDINT;	
END_VAR
VAR_OUTPUT
	OUT_Error				: BOOL;
	OUT_Busy				: BOOL;
	OUT_Result				: INT;
END_VAR
VAR
	Etape					: UINT;
	
	TrigStart				: R_TRIG;
	RsStart					: RS;
	bCreateTable			: BOOL;
	TrigCreateTable			: R_TRIG;
	RsCreateTable			: RS;
	PLCDBCreateEvt 			: FB_PLCDBCreateEvt(sNetID := '', tTimeout := T#5S);
	SqlLiteConf				: T_DBConfig_SQLite;
	DbFullDirName			: T_MAXSTRING;	
	sExtension				: STRING:= '.db';
	tcMessage    	 		: I_TcMessage;
	
	AX_ColArray				: ARRAY[0..3] OF ST_ColumnInfo;
	
	dBID_Test				: UDINT := 1;
	KK						: UDINT;
	bExisteDeja				: BOOL;	
END_VAR

OUT_Busy := TRUE;
AX_ColArray[0].sName := 'TimeStamp';     	AX_ColArray[0].eType := E_ColumnType.DateTime;   	AX_ColArray[0].nLength := 4;    
AX_ColArray[1].sName := 'TimeStamp_Ms';    	AX_ColArray[1].eType := E_ColumnType.Integer;    	AX_ColArray[1].nLength := 4;
AX_ColArray[2].sName := 'ParentId';   		AX_ColArray[2].eType := E_ColumnType.Integer;   	AX_ColArray[2].nLength := 4;
AX_ColArray[3].sName := 'Value';   			AX_ColArray[3].eType := E_ColumnType.Float;   		AX_ColArray[3].nLength := 8;


IF IN_DbType = 1 THEN
	sExtension := '.db';
ELSIF IN_DbType = 2 THEN
	sExtension := '.sdf';
END_IF

DbFullDirName := Concat(STR1:=Concat(STR1:= IN_Dir, STR2 := IN_Name), STR2 := sExtension);
SqlLiteConf.bAuthentification := FALSE;
SqlLiteConf.sServer := DbFullDirName;

FOR KK := 0 TO MAX_CONFIGURATIONS DO
	IF IN_ConfigDbActuelle[KK].sServer = DbFullDirName THEN
		bExisteDeja := TRUE;
		OUT_Result := -1;
		OUT_Busy := FALSE;
		OUT_Error := FALSE;
		bCreateTable := FALSE;
		IN_hDBID := IN_ConfigDbActuelle[KK].hDBID;
		EXIT;
	END_IF
	IF KK = MAX_CONFIGURATIONS THEN
		bExisteDeja := FALSE;
	END_IF
END_FOR

TrigStart(CLK := IN_Start AND NOT bExisteDeja);
RsStart(SET := TrigStart.Q);
IF RsStart.Q1 THEN
	IF PLCDBCreateEvt.Database(pDatabaseConfig := ADR(SqlLiteConf), cbDatabaseConfig := SIZEOF(SqlLiteConf), bCreateXMLConfig := TRUE, pDBID := ADR(dBID_Test)) THEN
		IF PLCDBCreateEvt.ipTcResult.nEventId = 59 THEN
			OUT_Error := FALSE;
			OUT_Result := -1;
			OUT_Busy := FALSE;	
			TrigStart(CLK := FALSE);
			bCreateTable := FALSE;
			Etape := 0;
			RsCreateTable(RESET1 := TRUE);
			RsCreateTable(RESET1 := FALSE);
		ELSIF PLCDBCreateEvt.bError THEN
			tcMessage := PLCDBCreateEvt.ipTcResult;
			OUT_Error := TRUE;
		ELSE
			Etape := 1;
			IN_hDBID := dBID_Test;
			bCreateTable := TRUE; 
		END_IF
		RsStart(RESET1 := TRUE);
		RsStart(RESET1 := FALSE);
	END_IF
END_IF

TrigCreateTable(CLK := bCreateTable);
RsCreateTable(SET:= TrigCreateTable.Q);

IF RsCreateTable.Q1 AND ETAPE = 1 THEN
	IF PLCDBCreateEvt.Table(hDBID := IN_hDBID, sTableName := IN_TableName,  pTableCfg := ADR(AX_ColArray), cbTableCfg := SIZEOF(AX_ColArray)  ) THEN
		IF PLCDBCreateEvt.bError THEN
			Etape := 255;
			OUT_Error := TRUE;
			OUT_Result := -2;
		ELSE
			IN_Start := FALSE;
			bCreateTable := FALSE;
			Etape := 0;
			OUT_Result := 1;
			RsCreateTable(RESET1 := TRUE);
			RsCreateTable(RESET1 := FALSE);
			TrigStart(CLK := False);
			OUT_Busy := FALSE;	
			OUT_Error := FALSE;
		END_IF
	END_IF
END_IF

IF Etape = 255 THEN
	Etape := 0;
	bCreateTable := FALSE;
	IN_Start := FALSE;
	OUT_Busy := FALSE;	
	RsCreateTable(RESET1 := TRUE);
	RsCreateTable(RESET1 := FALSE);
	
END_IF

END_PROGRAM

// ---- 00_FunctionsBlocks/Beckhoff/Database/SQLite/SQLite_DeleteConfDb_1.TcPOU
PROGRAM SQLite_DeleteConfDb_1
VAR_INPUT
	IN_DbType				: UINT:= 1; // 1:T_DBConfig_SQLite, 2:T_DBConfig_SQLCe
	IN_hDBID         		: UDINT;
	IN_Start				: BOOL;
	
END_VAR
VAR_OUTPUT
	OUT_Error				: BOOL;
	OUT_Busy				: BOOL;
END_VAR
VAR
	Etape					: UINT;
	
	TrigStart				: R_TRIG;
	RsStart					: RS;
	bDeleteTable			: BOOL;
	TrigDeleteFile			: R_TRIG;
	RsDeleteTable			: RS;
	fbConfigTcDBSrv   		: FB_ConfigTcDBSrvEvt (sNetID := '', tTimeout := T#5S);
	DbFullDirName			: T_MAXSTRING;	
	sExtension				: STRING:= '.db';
	tcMessage    	 		: I_TcMessage;
	
	

END_VAR

OUT_Busy := TRUE;

TrigStart(CLK := IN_Start);
RsStart(SET := TrigStart.Q);
IF RsStart.Q1 THEN
	IF fbConfigTcDBSrv.Delete(eTcDBSrvConfigType := E_TcDBSrvConfigType.Database, hConfigID := IN_hDBID) THEN
		IF fbConfigTcDBSrv.bError THEN
			tcMessage := fbConfigTcDBSrv.ipTcResult;
			OUT_Error := TRUE;
			OUT_Busy := FALSE;
			Etape := 255;
		ELSE 
			OUT_Busy := FALSE;
			OUT_Error := FALSE;
			Etape := 0;
		END_IF
		TrigStart(CLK := FALSE);
		RsStart(RESET1 := TRUE);
		RsStart(RESET1 := FALSE);
	END_IF
END_IF

IF Etape = 255 THEN
	Etape := 0;
	bDeleteTable := FALSE;
	IN_Start := FALSE;
	OUT_Busy := FALSE;	
	RsDeleteTable(RESET1 := TRUE);
	RsDeleteTable(RESET1 := FALSE);
	
END_IF

END_PROGRAM

// ---- 00_FunctionsBlocks/Beckhoff/Database/UnixTimestamp.TcPOU
FUNCTION_BLOCK UnixTimestamp
VAR_OUTPUT
    seconds: ULINT;
    milliseconds: ULINT;
END_VAR

VAR
    localSystemTime : FB_LocalSystemTime := ( bEnable := TRUE, dwCycle := 1 );
    getTimeZoneInformation : FB_GetTimeZoneInformation;
    timeZoneInformation : ST_TimeZoneInformation;
    specificLocalTimeToFileTime : FB_TzSpecificLocalTimeToFileTime;
    fileTime: T_FILETIME;
    onZerothSecondLastCycle : BOOL;
END_VAR

// Get local system time
localSystemTime();

// On the zeroth second of each minutesync timezone information
IF (timeZoneInformation.standardName = '' OR (localSystemTime.systemTime.wSecond = 0 AND NOT onZerothSecondLastCycle)) THEN
    getTimeZoneInformation(sNetID := '', bExecute := TRUE, tzInfo => timeZoneInformation);
END_IF;

// Convert local system time to unix timestamps
specificLocalTimeToFileTime(in := Tc2_Utilities.SYSTEMTIME_TO_FILETIME(localSystemTime.systemTime), tzInfo := timeZoneInformation, out => fileTime);
seconds := (SHL(DWORD_TO_ULINT(fileTime.dwHighDateTime), 32) + DWORD_TO_ULINT(fileTime.dwLowDateTime)) / 10000000 - 11644473600;
milliseconds := (SHL(DWORD_TO_ULINT(fileTime.dwHighDateTime), 32) + DWORD_TO_ULINT(fileTime.dwLowDateTime)) / 10000 - 11644473600000;

onZerothSecondLastCycle := localSystemTime.systemTime.wSecond = 0;

END_FUNCTION_BLOCK

// ---- 00_FunctionsBlocks/Beckhoff/DataProcessing/Compress/FUN_CompressCSV.TcPOU
PROGRAM FUN_CompressCSV
VAR_INPUT
	InDirectory 		: T_MaxString;
END_VAR
VAR_OUTPUT
END_VAR
VAR
	Directory1		: T_MaxString;
	Directory2		: T_MaxString;
	FB_Time 			: FB_LocalSystemTime;
	CompressFile	: FB_CompressFile;
	PreviousMonth 	: WORD := 12;
	PreviousYear 	: WORD := 2018;
	CalDirectory 	: T_MaxString;
	DirChange		: BOOL;
	bTest 			: BOOL;
	TimeStruct_Local : TIMESTRUCT;
END_VAR

FB_Time(sNetID := '', bEnable := TRUE, dwCycle := 1, dwOpt := 1, tTimeout := T#50MS, systemTime => TimeStruct_Local);
IF FB_TIME.bValid THEN 
	IF PreviousMonth <> TimeStruct_Local.wMonth THEN
		Directory1 := Concat(InDirectory, concat(WORD_TO_STRING(TimeStruct_Local.wYear), '\'));
		
		IF PreviousYear <> TimeStruct_Local.wYear THEN
			Directory1 := Concat(InDirectory, concat(WORD_TO_STRING(TimeStruct_Local.wYear-1), '\'));
			PreviousYear := TimeStruct_Local.wYear;
		END_IF
		
		Directory2 := Concat(Directory1, concat(WORD_TO_STRING(PreviousMonth), '\'));
		PreviousMonth := TimeStruct_Local.wMonth;
		DirChange := TRUE;
	END_IF

	
	IF DirChange THEN	
		bTest := TRUE;
		CompressFile(IN_Directory := Directory2);	
		DirChange := FALSE;
	END_IF
END_IF

END_PROGRAM

// ---- 00_FunctionsBlocks/Beckhoff/DataProcessing/Database/DataBase_V2.TcPOU
PROGRAM DataBase_V2
// Cette fois, plutôt qu'1 base avec 3 tables, faire 3 bases par jour (100ms, 1s, 1m)
// Nouvelle architecture : fichiers minute dans le même fichier qu'historisation, les autres dans Database
 
VAR
	ParamBaseDir					: T_MAXString := 'C:\TwinCAT\Functions\Database\SQLite\';
	ParamHistDir					: T_MaxString := 'C:\TwinCAT\Functions\Historisation\';
	
	ParamDbType						: UINT;
	                        		
	DBID_GLOBAL						: ARRAY[1..3] OF UDINT;
	DBID_ToDelete					: ARRAY[1..3] OF UDINT;
	
	bTest							: BOOL;
	
    AX_DirDB						: ARRAY[1..3] OF T_MaxString :=[ParamBaseDir, ParamBaseDir, ParamBaseDir] ;
	                   		
	MesAlarmCode 					: WORD;
	MesWarningCode					: WORD;
	// INIT
		
                            		
	// CheckConfig          		
		bCheckConfig				: BOOL := TRUE;
		TrigCheckConfig				: R_TRIG;
		TrigInit					: F_TRIG;
		RS_CheckConfig				: RS;
		                    		
		ConfigTcDBSrvEvt  			: FB_ConfigTcDBSrvEvt(sNetId := '', tTimeout:=T#5S);
		                    		
		aDBConfig         			: ARRAY[0..MAX_CONFIGURATIONS] OF ST_ConfigDB;
		aAutoGrpConfig    			: ARRAY[0..MAX_CONFIGURATIONS] OF ST_ConfigAutoLogGrp;
		AX_NameBase					: ARRAY[0..MAX_CONFIGURATIONS] OF T_MaxString;
		AX_hDBID					: ARRAY[0..MAX_CONFIGURATIONS] OF BOOL;
		AX_hDBIDNull				: ARRAY[0..MAX_CONFIGURATIONS] OF BOOL;
		                    		
		nDbCount          			: UDINT;
		nAutoGrpCount     			: UDINT;
		tcMessage         			: I_TcMessage;
	
	// DayTrig 
		Trig_CreateFolder			: R_TRIG;
		RS_CreateFolder				: RS;
		RS_CreateDbDay				: RS;
		RS_DeleteConf				: RS;
		RS_DeleteFiles				: RS;
		RS_CompressOldFiles			: RS;
		bDayTrig					: BOOL:= TRUE;
		bCreateDirErr				: BOOL;
		bCreateDbErr				: BOOL;
		bDeleteConfErr				: BOOL;
		bDeleteFileErr				: BOOL;
		bCompressFileErr			: BOOL;
		CreateDir					: FB_CreateDir_V2;
        AX_Name						: ARRAY[1..3] OF STRING;    
		DeleteFile30Days			: FB_DeleteFile;          
		DeleteFile3Days				: FB_DeleteFile;          
		StartProcess 				: NT_StartProcess;
		
	// CreateDb Init        		
		bCreateDb					: BOOL := TRUE;
		DbidCreated					: UDINT := 1;
		DbCreated_Trig				: F_TRIG;
		AX_ColArray					: ARRAY[0..3] OF ST_ColumnInfo;
	                            	
	// One hour has elapsed
		Trig1hour					: R_TRIG;
		Rs1hour						: RS;
		OldDBID						: UDINT := 1;
		bDbCreated					: BOOL;
		bDbDelete					: BOOL;
		sReqCmd						: T_MAXSTRING;
		
	// New day 
		TrigJour					: R_TRIG;
		RsJour						: RS;
		b1jourSpDoing				: BOOL;
		TimeStruct3days				: TIMESTRUCT;
		TimeStruct1month			: TIMESTRUCT;
		Requete						: T_MaxString;
		sTimeStamp1					: STRING(255);
		sTimeStamp2					: STRING(255);
		Format						: FB_FormatString;
	
		
	// Insert	
	SQLExpert_InsertBuffer_1s		: FB_SQLExpert_InsertBuffer;
	SQLExpert_InsertBuffer_1m		: FB_SQLExpert_InsertBuffer;
	SQLExpert_InsertBuffer_100ms	: FB_SQLExpert_InsertBuffer;

	TON_100ms						: TON;
	TON_1m							: TON;
	TON_1s							: TON;
	

	
	bInit 							: BOOL := TRUE;
	KK								: UDINT;
	LL								: UDINT := 1;

	bTest1 							: BOOL;
	bTest2 							: BOOL;
	
END_VAR

// Trigger pour détecter nouvelle journée -> lance un check config + DayTrig pour faire les proc stockées
TrigJour(CLK := CalLocalTimeStruct.wHour = 0);
bCheckConfig := TrigJour.Q;
Trig_CreateFolder(CLK := TrigJour.Q OR binit);
RS_CreateFolder(SET := Trig_CreateFolder.Q);

// Methode pour vérifier la configuration actuellement activée sur front montant de bCheckConfig
M_Checkconfig();

IF NOT bCheckConfig THEN
	M_DayTrig();
END_IF 

IF bInit THEN
	M_Init();
END_IF

M_AlarmManagement();
(*--------------------------------------------------------------------------------------------*)
(*--------------------------------------------------------------------------------------------*)
// ICI JE LANCE LES ADD BUFFER POUR LES 3 TABLES
IF NOT bInit THEN
	SQLExpert_InsertBuffer_100ms(NomTable := 'Table100ms', hDBID := DBID_GLOBAL[1]);
	SQLExpert_InsertBuffer_1s(NomTable := 'Table1s', hDBID := DBID_GLOBAL[2]);
	SQLExpert_InsertBuffer_1m(NomTable := 'Table1m', hDBID := DBID_GLOBAL[3]);
	
	
	TON_100ms(IN := NOT bInit, PT := T#100MS);
	IF TON_100ms.Q THEN
		FOR KK := 1 TO 100 DO
			SQLExpert_InsertBuffer_100ms.M_AddLine(InStruct := GVL_DataBaseStructures.AX_Struct_100ms[KK]);
		END_FOR
		TON_100ms(IN := FALSE);
		TON_100ms(IN := TRUE);
	END_IF
	
	TON_1s(IN := NOT bInit, PT := T#1S);
	IF TON_1s.Q THEN
		FOR KK := 1 TO 1000 DO
			SQLExpert_InsertBuffer_1s.M_AddLine(InStruct := GVL_DataBaseStructures.AX_Struct_1s[KK]);
		END_FOR
		TON_1s(IN := FALSE);
		TON_1s(IN := TRUE);
	END_IF
	
	TON_1m(IN := NOT bInit, PT := T#1M);
	IF TON_1m.Q THEN
		FOR KK := 1 TO 1000 DO
			SQLExpert_InsertBuffer_1m.M_AddLine(InStruct := GVL_DataBaseStructures.AX_Struct_1m[KK]);
		END_FOR
		TON_1m(IN := FALSE);
		TON_1m(IN := TRUE);
	END_IF	

END_IF
(*--------------------------------------------------------------------------------------------*)
(*--------------------------------------------------------------------------------------------*)

METHOD M_AlarmManagement : BOOL
VAR
		FB_AlarmCodeManager : FB_AlarmCodeManager;
END_VAR
FB_AlarmCodeManager
(
	bAlarm1 := bCreateDirErr,
	bAlarm2 := bCreateDbErr,
	bAlarm3 := bDeleteConfErr,
	bAlarm4 := bDeleteFileErr,
	bAlarm5 := bCompressFileErr,
	wAlarmCode => MesAlarmCode
);
END_METHOD

METHOD M_CheckConfig : BOOL
VAR_INPUT
END_VAR
TrigCheckConfig(CLK := bCheckConfig OR binit);
RS_CheckConfig(SET := TrigCheckConfig.Q);
	
IF RS_CheckConfig.Q1 THEN
	IF ConfigTcDBSrvEvt.Read(
		pDBConfig := ADR(aDBConfig), 
		cbDBConfig := SIZEOF(aDBConfig), 
		pAutologGrpConfig := ADR(aAutoGrpConfig),
		cbAutoLogGrpConfig := SIZEOF(aAutoGrpConfig),
		pDBCount := ADR(nDbCount),
		pAutoLogGrpCount := ADR(nAutoGrpCount))
	 THEN
		IF ConfigTcDBSrvEvt.bError THEN
			tcMessage := ConfigTcDBSrvEvt.ipTcResult;
			bCheckConfig := FALSE; 
		ELSE
			bCheckConfig := FALSE; 
			FOR KK := 0 TO MAX_CONFIGURATIONS DO
				AX_hDBID[aDBConfig[KK].hDBID] := aDBConfig[KK].hDBID <> 0;
				AX_NameBase[KK] :=  aDBConfig[KK].sName;
			END_FOR
		END_IF  
		TrigCheckConfig(CLK := FALSE OR binit);
		RS_CheckConfig(RESET1 := TRUE);
		RS_CheckConfig(RESET1 := FALSE);
	END_IF
END_IF
END_METHOD

METHOD M_DayTrig : BOOL
VAR_INPUT
END_VAR
VAR
	DirTemp			: ARRAY[1..3] OF T_MaxString;
	AX_NameTemp		: ARRAY[1..3] OF STRING := ['Table100ms', 'Table1s', 'Table1m']; 	
	Dir30Days		: T_MaxString;
	Dir3Days		: T_MaxString; 	
	Dir3DaysComp1	: T_MaxString; 	
	Dir3DaysComp2	: T_MaxString; 	

	
END_VAR



TimeStruct3days := DT_TO_SYSTEMTIME( SYSTEMTIME_TO_DT (CalLocalTimeStruct) - T#3D);
TimeStruct1month := DT_TO_SYSTEMTIME( SYSTEMTIME_TO_DT (CalLocalTimeStruct) - T#30D);

// D'abord je commence par créer tous les dossiers
IF RS_CreateFolder.Q1 THEN
	DirTemp[1] := ParamHistDir;
	DirTemp[2] := Concat(STR1 := Concat(STR1 := ParamHistDir, STR2 := WORD_TO_STRING(CalLocalTimeStruct.wYear)), STR2 := '\');
	DirTemp[3] := CONCAT(STR1 := CONCAT(STR1 := Concat(STR1 := Concat(STR1 := ParamHistDir, STR2 := WORD_TO_STRING(CalLocalTimeStruct.wYear)), STR2 := '\'), STR2 := WORD_TO_STRING(CalLocalTimeStruct.wMonth)), STR2 := '\');
	
	AX_DirDB[1] := ParamBaseDir;
	AX_DirDB[2] := ParamBaseDir;
	AX_DirDB[3] := DirTemp[3];
	FOR KK := 1 TO 3 DO 
		AX_Name[KK] := CONCAT(STR1 := CONCAT(STR1 := CONCAT(STR1 := CONCAT(STR1 := CONCAT(STR1 := Concat(STR1 := WORD_TO_STRING(CalLocalTimeStruct.wYear), STR2 := ''), STR2 := WORD_TO_STRING(CalLocalTimeStruct.wMonth)), STR2:= ''), STR2:= WORD_TO_STRING(CalLocalTimeStruct.wDay)), STR2:= '_'), STR2:= AX_NameTemp[KK]);
	END_FOR
	
	IF LL < 4 THEN
		CreateDir(InPath := DirTemp[LL], InExe := LL < 4);
		IF NOT CreateDir.OutBusy THEN
			IF CreateDir.OutError AND NOT CreateDir.OutErrorId =1827 (*Dossier existe déjà*) THEN
				CreateDir(InExe := FALSE);
				bCreateDirErr := TRUE;
			ELSE
				bCreateDirErr := FALSE;
				CreateDir(InExe := FALSE);
				LL := LL + 1;
			END_IF
			CreateDir(InPath := DirTemp[LL], InExe := FALSE);
		END_IF
	ELSE
		RS_CreateFolder(RESET1 := TRUE);
		RS_CreateFolder(RESET1 := FALSE);
		RS_CreateDbDay(SET := TRUE);
		RS_CreateDbDay(SET := FALSE);
		LL := 1;
	END_IF
END_IF

// Ensuite je créée les bases 
IF RS_CreateDbDay.Q1 THEN
	IF LL < 4 THEN
		SQLite_CreateDb_V2(IN_DbType := 1, IN_Dir := AX_DirDB[LL],IN_Name := AX_Name[LL], IN_TableName := AX_NameTemp[LL], IN_hDBID := DBID_GLOBAL[LL], IN_Start := bCreateDb, IN_ConfigDbActuelle := aDBConfig);
		IF NOT SQLite_CreateDb_V2.OUT_Busy THEN
			SQLite_CreateDb_V2(IN_Start := FALSE, IN_hDBID := DBID_GLOBAL[LL]);
			IF SQLite_CreateDb_V2.OUT_Error THEN
				SQLite_CreateDb_V2(IN_Start := FALSE, IN_hDBID := DBID_GLOBAL[LL]);
				bCreateDbErr := TRUE;
			ELSE
				SQLite_CreateDb_V2(IN_Start := FALSE, IN_hDBID := DBID_GLOBAL[LL]);
				LL := LL + 1;
				bCreateDbErr := FALSE;
			END_IF
		END_IF
	ELSE
		LL := 1;
		RS_CreateDbDay(RESET1 := TRUE);
		RS_CreateDbDay(RESET1 := FALSE);
		RS_DeleteConf(SET := TRUE AND NOT bInit);
		RS_DeleteConf(SET := FALSE);
		bDayTrig := False;
	END_IF
END_IF

// Ensuite je supprime les vieilles tables de la conf précédente
IF RS_DeleteConf.Q1 THEN
	IF LL < 4 THEN
		DBID_ToDelete[LL] := SEL(DBID_GLOBAL[LL] = LL, LL, LL+3);
		// CELA NE SUPPRIME QUE LES CONFS
		SQLite_DeleteConfDb(IN_DbType := 1, IN_hDBID := DBID_ToDelete[LL], IN_Start := TRUE);
		IF NOT SQLite_DeleteConfDb.OUT_Busy THEN
			IF SQLite_DeleteConfDb.OUT_Error THEN
				SQLite_DeleteConfDb(IN_Start := FALSE);
				bDeleteConfErr := TRUE;
			ELSE
				bDeleteConfErr := FALSE;
				SQLite_DeleteConfDb(IN_Start := FALSE);
				LL := LL + 1;
			END_IF
		END_IF
	ELSE
		LL := 1;
		RS_DeleteConf(RESET1 := TRUE);
		RS_DeleteConf(RESET1 := FALSE);
		RS_DeleteFiles(SET := TRUE);
		RS_DeleteFiles(SET := FALSE);
	END_IF
END_IF

// Et enfin, je supprime les vieux fichiers : plus de 30 jours pour les 1s, plus de 3 jours pour les 100ms
IF RS_DeleteFiles.Q1 THEN
	Dir30Days := CONCAT(STR1:=CONCAT(STR1:=CONCAT(STR1 := CONCAT(STR1 := CONCAT(STR1 := CONCAT(STR1 := CONCAT(STR1 := Concat(STR1 := ParamBaseDir, STR2 := WORD_TO_STRING(TimeStruct1month.wYear)), STR2 := ''), STR2 := WORD_TO_STRING(TimeStruct1month.wMonth)), STR2:= ''), STR2:= WORD_TO_STRING(TimeStruct1month.wDay)), STR2:= '_'), STR2:= AX_NameTemp[LL]), STR2 := '.db');
	Dir3Days := CONCAT(STR1:=CONCAT(STR1:=CONCAT(STR1 := CONCAT(STR1 := CONCAT(STR1 := CONCAT(STR1 := CONCAT(STR1 := Concat(STR1 := ParamBaseDir, STR2 := WORD_TO_STRING(TimeStruct3days.wYear)), STR2 := ''), STR2 := WORD_TO_STRING(TimeStruct3days.wMonth)), STR2:= ''), STR2:= WORD_TO_STRING(TimeStruct3days.wDay)), STR2:= '_'), STR2:= AX_NameTemp[LL]), STR2 := '.db');
	
	DeleteFile30Days(IN_Dir := Dir30Days, IN_Start := TRUE);
	DeleteFile3Days(IN_Dir := Dir3Days, IN_Start := TRUE);
	
	IF NOT DeleteFile3Days.OUT_Busy AND NOT DeleteFile30Days.OUT_Busy AND LL < 2 THEN
		IF NOT DeleteFile30Days.OUT_Error AND NOT DeleteFile3Days.OUT_Error THEN
			LL := LL + 1;
			DeleteFile30Days(IN_Start := FALSE);
			DeleteFile3Days(IN_Start := FALSE);
			bDeleteFileErr := FALSE;
		ELSE
			bDeleteFileErr := TRUE;
			DeleteFile30Days(IN_Start := FALSE);
			DeleteFile3Days(IN_Start := FALSE);
		END_IF
	ELSIF NOT DeleteFile3Days.OUT_Busy AND NOT DeleteFile30Days.OUT_Busy AND LL = 2 THEN
		IF NOT DeleteFile30Days.OUT_Error AND NOT DeleteFile3Days.OUT_Error THEN
			LL := 1;
			bDeleteFileErr := FALSE;
			DeleteFile30Days(IN_Start := FALSE);
			DeleteFile3Days(IN_Start := FALSE);
			RS_DeleteFiles(reset1 := TRUE);
			RS_DeleteFiles(reset1 := FALSE);
			RS_CompressOldFiles(set := TRUE);
			RS_CompressOldFiles(Set := FALSE);
		ELSE
			bDeleteFileErr := TRUE;
			DeleteFile30Days(IN_Start := FALSE);
			DeleteFile3Days(IN_Start := FALSE);
		END_IF
	END_IF
END_IF

IF RS_CompressOldFiles.Q1 THEN
	Dir3DaysComp1 := CONCAT(STR1:=CONCAT(STR1:=CONCAT(STR1 := CONCAT(STR1 := CONCAT(STR1 := CONCAT(STR1 := CONCAT(STR1 := Concat(STR1 := ParamBaseDir, STR2 := WORD_TO_STRING(TimeStruct3days.wYear)), STR2 := ''), STR2 := WORD_TO_STRING(TimeStruct3days.wMonth)), STR2:= ''), STR2:= WORD_TO_STRING(TimeStruct3days.wDay)), STR2:= '_'), STR2:= AX_NameTemp[1]), STR2 := '.db');
	Dir3DaysComp2 := CONCAT(STR1:=CONCAT(STR1:=CONCAT(STR1 := CONCAT(STR1 := CONCAT(STR1 := CONCAT(STR1 := CONCAT(STR1 := Concat(STR1 := ParamBaseDir, STR2 := WORD_TO_STRING(TimeStruct3days.wYear)), STR2 := ''), STR2 := WORD_TO_STRING(TimeStruct3days.wMonth)), STR2:= ''), STR2:= WORD_TO_STRING(TimeStruct3days.wDay)), STR2:= '_'), STR2:= AX_NameTemp[2]), STR2 := '.db');
	StartProcess
	(
		NETID := '',
		PATHSTR := 'C:\Windows\System32\compact.exe',
		DIRNAME := 'C:\Windows\System32',
		COMNDLINE :=  CONCAT(STR1:=CONCAT(STR1:=CONCAT(STR1:=CONCAT(STR1:=' /c "',STR2:=Dir3DaysComp1), str2:='"  "'), STR2:=Dir3DaysComp2),str2:='"'),
		Start := RS_CompressOldFiles.Q1,
		TMOUT := T#3M
	);
	IF NOT StartProcess.BUSY THEN
		IF NOT StartProcess.ERR THEN
			StartProcess(Start := FALSE);
			bCompressFileErr := FALSE;
			RS_CompressOldFiles(RESET1:= TRUE);
			RS_CompressOldFiles(RESET1:= FALSE);
		ELSE
			StartProcess(Start := FALSE);
			bCompressFileErr := TRUE;
		END_IF
	END_IF	
END_IF
END_METHOD

METHOD M_Init : BOOL
VAR_INPUT
END_VAR


bInit := (bCheckConfig) OR (bDayTrig);
END_METHOD

END_PROGRAM

// ---- 00_FunctionsBlocks/Beckhoff/DataProcessing/Database/FB_DeleteFile.TcPOU
FUNCTION_BLOCK FB_DeleteFile
VAR_INPUT
	IN_Start				: BOOL;
	IN_Dir					: T_MaxString;
END_VAR
VAR_OUTPUT
	OUT_Error				: BOOL;
	OUT_Busy				: BOOL;
END_VAR
VAR
	
	TrigStart				: R_TRIG;
	RsStart					: RS;
	FileDelete				: FB_FileDelete;
	
	

END_VAR

OUT_Busy := TRUE;

TrigStart(CLK := IN_Start);
FileDelete(sNetId := '', sPathName := IN_Dir, bExecute := TrigStart.Q);

RsStart(SET := TrigStart.Q);
IF RsStart.Q1 THEN
	IF NOT FileDelete.bBusy THEN
		IF FileDelete.bError THEN
			OUT_Error := TRUE;
			OUT_Busy := FALSE;
		ELSE 
			OUT_Error := FALSE;
			OUT_Busy := FALSE;
		END_IF
		TrigStart(CLK := FALSE);
		RsStart(RESET1 := TRUE);
		RsStart(RESET1 := FALSE);
	END_IF
END_IF

END_FUNCTION_BLOCK

// ---- 00_FunctionsBlocks/Beckhoff/DataProcessing/Database/FB_SQLExpert_InsertBuffer.TcPOU
FUNCTION_BLOCK FB_SQLExpert_InsertBuffer
// Fonctionnement : Tableau de 2000 structures en input. Dès qu'on atteint 1000 structures remplies, décalage de l'espace mémoire
// pour en 1 temps de cycle pour ne pas perdre de données sur le transfert.
VAR CONSTANT
	CstNbLigneBuffer		: DINT:= 250;
	CstNbLigneBufferMax	 	: DINT:= 5000;

END_VAR

VAR_INPUT
	NomTable				: STRING := 'Table100ms';
	hDBID					: UDINT;
END_VAR

VAR_OUTPUT
	OUT_Error				: BOOL;
	OUT_Busy				: BOOL;
END_VAR

VAR
	ETAPE					: UINT;

    myStruct      			: ARRAY[1..CstNbLigneBuffer] OF St_DataHisto;
	myStructMax    			: ARRAY[1..CstNbLigneBufferMax] OF St_DataHisto;
	StructNull				: St_DataHisto;

    SQLDatabase				: FB_SQLDatabaseEvt('',T#10S);
	SQLCommand1				: FB_SQLCommandEvt('',T#10S);
	SQLCommandNull			: FB_SQLCommandEvt('',T#10S);
	bConnected				: BOOL;              	        	

	TrameValues				: T_MaxString := ' ([Timestamp],[Timestamp_Ms],[ParentId],[Value])';
	pPosRequete				: DINT;                		
	RequeteFinale			: ARRAY[1..100] OF STRING(1000);	
	RequeteFinaleNull		: ARRAY[1..100] OF STRING(1000);	
	sTimeStamp				: STRING(255);               	
	RequeteEntete			: STRING(1000);
	sInsertValue			: STRING(1000);
	Format					: FB_FormatString;
	                		
	NbElemBuffer			: DINT;
	KK						: DINT;
	                    	
	CmdStart				: BOOL;
	TrigCmdExec				: R_TRIG;
	TrigStart				: R_TRIG;
	RsStart					: RS;
	
	// Insert
		hDBID_BaseTampon	: UINT := 3;
	// AlarmManagement      
		bBufferMaxFull 		: BOOL;        		
		bInStructNull		: BOOL;
		
		
		
	
END_VAR

NbElemBuffer := M_Count();
CmdStart := NbElemBuffer>= CstNbLigneBuffer;


TrigStart(CLK := CmdStart);
IF TrigStart.Q THEN
	FOR KK := 1 TO CstNbLigneBuffer DO
		myStruct[KK] := myStructMax[KK];
	END_FOR
END_IF


// call functionblock

CASE ETAPE OF
	0://INITIALISATION  & CONNECTION
		RequeteEntete := concat(concat('INSERT INTO ',NomTable),concat(TrameValues,' VALUES '));
		RsStart(SET := TrigStart.Q);
		IF RsStart.Q1 THEN
			IF SQLDatabase.Connect(hDBID := hDBID) THEN;
				bConnected := NOT sqldatabase.bError;
				IF bConnected THEN
					ETAPE := 1;
				ELSE
					ETAPE := 255;
				END_IF
			END_IF
		END_IF
		
	1: // CONNECTED
		IF SQLDatabase.CreateCmd(pSQLCommand := ADR(SQLCommand1)) THEN 
			IF NOT SQLCommand1.bError THEN
				ETAPE := 2;
			ELSIF SQLCommand1.bError THEN
				ETAPE := 255;
			END_IF
		END_IF
	2:
		MEMCPY(srcAddr:= ADR(RequeteEntete), destAddr := ADR(requeteFinale), n:= SIZEOF(RequeteEntete));
		pPosRequete := LEN(STR := RequeteEntete);
		FOR KK:= 1 TO CstNbLigneBuffer-1 DO
			sTimeStamp	:= right(STR := DT_TO_STRING(myStruct[KK].Timestamp), SIZE := LEN(DT_TO_STRING(myStruct[KK].Timestamp))-3);
			Format(sFormat := '($'%s $',%.3d,%.4d,%5.2f),', arg1 := F_STRING(sTimeStamp),arg2:=F_DINT(myStruct[KK].Timestamp_Ms), arg3:= F_DINT(myStruct[KK].ParentId), arg4:= F_LREAL(myStruct[KK].Value), sOut=>sInsertValue);
			MEMCPY(srcAddr:= ADR(sInsertValue), destAddr := ADR(requeteFinale)+DINT_TO_DWORD(pPosRequete), n:= SIZEOF(sInsertValue));
			pPosRequete:= pPosRequete + LEN(STR := sInsertValue);
		END_FOR
		sTimeStamp	:= right(STR := DT_TO_STRING(myStruct[KK].Timestamp), SIZE := LEN(DT_TO_STRING(myStruct[KK].Timestamp))-3);
		Format(sFormat := '($'%s $',%.3d,%.4d,%5.2f)', arg1 := F_STRING(sTimeStamp),arg2:=F_DINT(myStruct[KK].Timestamp_Ms), arg3:= F_DINT(myStruct[KK].ParentId), arg4:= F_LREAL(myStruct[KK].Value), sOut=>sInsertValue);
		MEMCPY(srcAddr:= ADR(sInsertValue), destAddr := ADR(requeteFinale)+DINT_TO_DWORD(pPosRequete), n:= SIZEOF(sInsertValue));
	
		IF SQLCommand1.Execute(pSQLCmd := ADR(RequeteFinale), cbSQLCmd := SIZEOF(Requetefinale))THEN
			
			IF  NOT SQLCommand1.bError THEN
				ETAPE := 3;
			ELSIF SQLCommand1.bError THEN
				ETAPE := 255;
			END_IF
		END_IF
	3:
			IF SQLDatabase.Disconnect() THEN
				ETAPE := 4;
			END_IF 
	4:
		IF NOT SQLDatabase.bError THEN
			RequeteFinale := RequeteFinaleNull;
			FOR KK := CstNbLigneBuffer TO CstNbLigneBufferMax -1 DO
				myStructMax[KK+1-CstNbLigneBuffer]:= myStructMax[KK+1];
			END_FOR
			
			FOR KK := CstNbLigneBufferMax-CstNbLigneBuffer+1 TO CstNbLigneBufferMax DO
				myStructMax[KK]:= StructNull;
			END_FOR			
			
			TrigStart(CLK := FALSE);
			RsStart(RESET1 := TRUE);
			RsStart(RESET1 := FALSE);
			TrigCmdExec(CLK := FALSE);
			CmdStart := FALSE;
			Etape := 0;
			OUT_Error := FALSE;
		ELSE 
			ETAPE := 255;
		END_IF
	255: 
		RequeteFinale := RequeteFinaleNull;
		OUT_Error := TRUE;
		Etape := 0;
		RsStart(RESET1 := TRUE);
		RsStart(RESET1 := FALSE);
		TrigCmdExec(CLK := FALSE);
		CmdStart := FALSE;
		
END_CASE

METHOD M_AddLine : BOOL
VAR_INPUT
	InStruct			: St_DataHisto;
END_VAR

VAR
END_VAR
// Check the biggest buffer isn't full
IF MEMCMP(pBuf1 := ADR(StructNull), pBuf2 := ADR(myStructMax[CstNbLigneBufferMax]), n := SIZEOF(StructNull)) <> 0 THEN
	bBufferMaxFull := TRUE;
ELSE
	//Check the input struct isn't null
	IF MEMCMP(pBuf1 := ADR(StructNull), pBuf2 := ADR(InStruct), n := SIZEOF(StructNull)) = 0 THEN
		bInStructNull := TRUE;
	ELSE
		// We parse the biggest buffer
		FOR KK := 1 TO CstNbLigneBufferMax DO 
			IF MEMCMP(pBuf1 := ADR(StructNull), pBuf2 := ADR(myStructMax[KK]), n := SIZEOF(StructNull)) = 0 THEN
				myStructMax[KK] := InStruct;
				bBufferMaxFull := FALSE;
				EXIT;
			END_IF
		END_FOR
	END_IF
END_IF
END_METHOD

METHOD M_AlarmManager : BOOL
VAR_INPUT
	AlarmCode : WORD;
	
END_VAR


AlarmCode.0 := bBufferMaxFull;
AlarmCode.1 := bInStructNull;
END_METHOD

METHOD M_Count : DINT
VAR_INPUT
END_VAR
VAR

END_VAR
FOR KK := 1 TO CstNbLigneBufferMax DO 

	IF MEMCMP(pBuf1 := ADR(StructNull), pBuf2 := ADR(myStructMax[KK]), n := SIZEOF(StructNull)) = 0 THEN
		EXIT ;
	END_IF
END_FOR

M_Count := MIN(KK, CstNbLigneBufferMax);
END_METHOD

END_FUNCTION_BLOCK

